		(*-----------------------Weiterschaltbedingungen----------------------------*)
		IF zyl_bawe_vorschub.st_ctrl.out.b_ausgefahren AND gb_ba_auto_kontroller THEN
			zyl_bawe_vorschub.st_ctrl.in.b_ausfahren := FALSE;
			IF i16_akt_einfaedeln < i16_vorgabe_einfaedeln THEN
				fb_state_entry.i16_next_step := 640;
			ELSE
				fb_state_entry.i16_next_step := 690; (*mit Wartezeit alt auf 700*)
			END_IF
		END_IF

(*=======================================================*)
	640:	(* Halter links ausfahren *)
		IF fb_state_entry.E THEN
			zyl_bawe_halter_li.st_ctrl.in.b_ausfahren := TRUE;
		END_IF

		(*-----------------------Weiterschaltbedingungen----------------------------*)
		IF zyl_bawe_halter_li.st_ctrl.out.b_ausgefahren AND gb_ba_auto_kontroller THEN
			zyl_bawe_halter_li.st_ctrl.in.b_ausfahren := FALSE;
			fb_state_entry.i16_next_step := 650;
		END_IF

(*=======================================================*)
	650:	(* Fänger links einfahren *)
		IF fb_state_entry.E THEN
			zyl_bawe_faenger_li.st_ctrl.in.b_einfahren := TRUE;
		END_IF

		(*-----------------------Weiterschaltbedingungen----------------------------*)
		IF zyl_bawe_faenger_li.st_ctrl.out.b_eingefahren AND gb_ba_auto_kontroller THEN
			zyl_bawe_faenger_li.st_ctrl.in.b_einfahren := FALSE;
			fb_state_entry.i16_next_step := 660;
		END_IF

(*=======================================================*)
	660:	(* Vorschub einfahren *)
		IF fb_state_entry.E THEN
			zyl_bawe_vorschub.st_ctrl.in.b_einfahren := TRUE;
		END_IF

		(*-----------------------Weiterschaltbedingungen----------------------------*)
		IF zyl_bawe_vorschub.st_ctrl.out.b_eingefahren AND gb_ba_auto_kontroller THEN
			zyl_bawe_vorschub.st_ctrl.in.b_einfahren := FALSE;
			fb_state_entry.i16_next_step := 670;
		END_IF

(*=======================================================*)
	670:	(* Fänger links ausfahren *)
		IF fb_state_entry.E THEN
			zyl_bawe_faenger_li.st_ctrl.in.b_ausfahren := TRUE;
		END_IF

		(*-----------------------Weiterschaltbedingungen----------------------------*)
		IF zyl_bawe_faenger_li.st_ctrl.out.b_ausgefahren AND gb_ba_auto_kontroller THEN
			zyl_bawe_faenger_li.st_ctrl.in.b_ausfahren := FALSE;
			fb_state_entry.i16_next_step := 680;
		END_IF

(*=======================================================*)
	680:	(* Halter links einfahren *)
		IF fb_state_entry.E THEN
			zyl_bawe_halter_li.st_ctrl.in.b_einfahren := TRUE;
		END_IF

		(*-----------------------Weiterschaltbedingungen----------------------------*)
		IF zyl_bawe_halter_li.st_ctrl.out.b_eingefahren AND gb_ba_auto_kontroller THEN
			zyl_bawe_halter_li.st_ctrl.in.b_einfahren := FALSE;
			fb_state_entry.i16_next_step := 630;
		END_IF
(*=======================================================*)
	690:	(* Wartezeit damit der Fänger vom WZ trifft*)
		IF	 fb_state_entry.E THEN
			fb_ton_wz.IN:=FALSE;
		END_IF
		fb_ton_wz(IN:=TRUE,PT:=t#1000ms);
		(*-----------------------Weiterschaltbedingungen----------------------------*)
		IF 	fb_ton_wz.Q THEN
			fb_ton_wz.IN:=FALSE;
			fb_state_entry.i16_next_step := 700;
		END_IF

(*=======================================================*)
	700:	(* Nocken für Zylinder am Bandeinzug einschalten und somit Bandfänger ausfahren bzw. Bremse an Servobandeinzug wieder fest machen. *)
		CASE gst_datensatz.st_wkz.i16_typ_bandeinzug OF

			BANDWECHSLER_V2:

				IF fb_state_entry.E THEN
					(* Bandwechsler V2 ohne Sensoren und anderen Zylindern *)
					gst_datensatz.st_wkz.nockenschaltwerk_bestueckachse.arr_nocken[NO_BW_BANDFAENGER_BAWEV2_EINFAHREN].b_camvalid := TRUE;
					gst_datensatz.st_wkz.nockenschaltwerk_bestueckachse.arr_nocken[NO_BW_BANDFAENGER_BAWEV2_AUSFAHREN].b_camvalid := TRUE;
					gst_datensatz.st_wkz.nockenschaltwerk_bestueckachse.arr_nocken[NO_BW_BANDKLEMMEN_BAWEV2_EINFAHREN].b_camvalid := TRUE;
					gst_datensatz.st_wkz.nockenschaltwerk_bestueckachse.arr_nocken[NO_BW_BANDKLEMMEN_BAWEV2_AUSFAHREN].b_camvalid := TRUE;

					gst_datensatz.st_wkz.nockenschaltwerk_bestueckachse.arr_nocken[NO_PNEUMATIKBANDEINZUG_GLS].b_camvalid := TRUE;

					zyl_bandfaenger.fb.b_no_gesteuert_im_norm_betrieb := FALSE;
					zyl_bandklemmen.fb.b_no_gesteuert_im_norm_betrieb := FALSE;
					fb_ton_wz.PT := t#500ms;
					fb_ton_wz.IN := TRUE;
				END_IF
		
				(*-----------------------Weiterschaltbedingungen----------------------------*)
				IF fb_ton_wz.Q THEN
					fb_ton_wz.IN := FALSE;
					fb_state_entry.i16_next_step := 710;
				END_IF

			SERVO:
				IF fb_state_entry.E THEN
					axis_bandeinzug_achse.st_ctrl.in.b_bremse_auf := TRUE;	(* Bremse auf zum Position übernehmen *)
				END_IF

				(*-----------------------Weiterschaltbedingungen----------------------------*)
				IF axis_bandeinzug_achse.st_ctrl.out.b_bremse_geoeffnet THEN
					axis_bandeinzug_achse.st_ctrl.in.b_bremse_auf := FALSE;
					fb_state_entry.i16_next_step := 710;
				END_IF
		END_CASE;

(*=======================================================*)
	710:	(* Fänger links einfahren *)
		IF fb_state_entry.E THEN
			zyl_bawe_faenger_li.st_ctrl.in.b_einfahren := TRUE;
		END_IF

		(*-----------------------Weiterschaltbedingungen----------------------------*)
		IF zyl_bawe_faenger_li.st_ctrl.out.b_eingefahren
		AND gb_ba_auto_kontroller THEN
			zyl_bawe_faenger_li.st_ctrl.in.b_einfahren := FALSE;
			(* Bandwechsel ist fertig *)
			st_ctrl_out.b_fertig := TRUE;
			fb_state_entry.i16_next_step := BEREIT;
		END_IF

(*=======================================================*)
	FEHLER:
		IF fb_state_entry.E THEN
			st_ctrl_out.b_fehler := TRUE;
			fb_ton_quitt.IN := FALSE;
			zyl_bawe_vorschub.st_ctrl.in.b_quittieren := FALSE;
			zyl_bawe_querschub.st_ctrl.in.b_quittieren := FALSE;
			zyl_bawe_faenger_li.st_ctrl.in.b_quittieren := FALSE;
			zyl_bawe_faenger_re.st_ctrl.in.b_quittieren := FALSE;
			zyl_bawe_halter_li.st_ctrl.in.b_quittieren := FALSE;
			zyl_bawe_halter_re.st_ctrl.in.b_quittieren := FALSE;
			zyl_haspel_verschieben.st_ctrl.in.b_quittieren := FALSE;
			zyl_bandeinzuege_verschieben.st_ctrl.in.b_quittieren := FALSE;
		END_IF

		(*-----------------------Weiterschaltbedingungen----------------------------*)
		IF st_ctrl_in.b_quitt AND NOT fb_state_entry.E THEN
			st_ctrl_out.b_fehler := TRUE;
			zyl_bawe_vorschub.st_ctrl.in.b_quittieren := TRUE;
			zyl_bawe_querschub.st_ctrl.in.b_quittieren := TRUE;
			zyl_bawe_faenger_li.st_ctrl.in.b_quittieren := TRUE;
			zyl_bawe_faenger_re.st_ctrl.in.b_quittieren := TRUE;
			zyl_bawe_halter_li.st_ctrl.in.b_quittieren := TRUE;
			zyl_bawe_halter_re.st_ctrl.in.b_quittieren := TRUE;
			zyl_haspel_verschieben.st_ctrl.in.b_quittieren := TRUE;
			zyl_bandeinzuege_verschieben.st_ctrl.in.b_quittieren := TRUE;
			fb_ton_quitt.IN := TRUE;
		END_IF

		IF fb_ton_quitt.Q THEN
			fb_ton_quitt.IN := FALSE;
			fb_state_entry.i16_next_step := INIT;
		END_IF

(*=======================================================*)
	STOP:
		IF fb_state_entry.E THEN
			fb_ton_quitt.IN := FALSE;
			zyl_bawe_vorschub.st_ctrl.in.b_quittieren := FALSE;
			zyl_bawe_querschub.st_ctrl.in.b_quittieren := FALSE;
			zyl_bawe_faenger_li.st_ctrl.in.b_quittieren := FALSE;
			zyl_bawe_faenger_re.st_ctrl.in.b_quittieren := FALSE;
			zyl_bawe_halter_li.st_ctrl.in.b_quittieren := FALSE;
			zyl_bawe_halter_re.st_ctrl.in.b_quittieren := FALSE;
			zyl_haspel_verschieben.st_ctrl.in.b_quittieren := FALSE;
			zyl_bandeinzuege_verschieben.st_ctrl.in.b_quittieren := FALSE;
		END_IF

		(*-----------------------Weiterschaltbedingungen----------------------------*)
		IF st_ctrl_in.b_quitt AND NOT fb_state_entry.E THEN
			fb_ton_quitt.IN := TRUE;
			zyl_bawe_vorschub.st_ctrl.in.b_quittieren := TRUE;
			zyl_bawe_querschub.st_ctrl.in.b_quittieren := TRUE;
			zyl_bawe_faenger_li.st_ctrl.in.b_quittieren := TRUE;
			zyl_bawe_faenger_re.st_ctrl.in.b_quittieren := TRUE;
			zyl_bawe_halter_li.st_ctrl.in.b_quittieren := TRUE;
			zyl_bawe_halter_re.st_ctrl.in.b_quittieren := TRUE;
			zyl_haspel_verschieben.st_ctrl.in.b_quittieren := TRUE;
			zyl_bandeinzuege_verschieben.st_ctrl.in.b_quittieren := TRUE;
		END_IF

		IF fb_ton_quitt.Q THEN
			fb_ton_quitt.IN := FALSE;
			fb_state_entry.i16_next_step := INIT;
		END_IF
END_CASE

fb_state_entry(
	i16_next_step:= , 
	i16_pos:= 2,
	s_debugtext:= ,
	E=> ,
	X=> , 
	i16_step=> ,
	i16_last_step=> );

IF st_config.b_config_fertig THEN
	(* Fehlermeldungen und Betriebsmeldungen ab dem Startindex in die globalen Meldungsarrays schreiben *)
	garr_stoermeldungen[st_config.i16_meld_startindex + 0] := sm_halter_nicht_oben;
	garr_stoermeldungen[st_config.i16_meld_startindex + 1] := sm_bandwechsel_ohne_ende;
	garr_stoermeldungen[st_config.i16_meld_startindex + 2] := sm_kein_band_anderer_einzug;
	garr_stoermeldungen[st_config.i16_meld_startindex + 3] := sm_kein_band_in_akt_einzug;
	garr_stoermeldungen[st_config.i16_meld_startindex + 4] := FALSE;
	garr_stoermeldungen[st_config.i16_meld_startindex + 5] := FALSE;
	garr_stoermeldungen[st_config.i16_meld_startindex + 6] := FALSE;
	garr_stoermeldungen[st_config.i16_meld_startindex + 7] := FALSE;
	garr_stoermeldungen[st_config.i16_meld_startindex + 8] := FALSE;
	garr_stoermeldungen[st_config.i16_meld_startindex + 9] := FALSE;
	garr_stoermeldungen[st_config.i16_meld_startindex + 10] := FALSE;
	garr_stoermeldungen[st_config.i16_meld_startindex + 11] := FALSE;
	garr_stoermeldungen[st_config.i16_meld_startindex + 12] := FALSE;
	garr_stoermeldungen[st_config.i16_meld_startindex + 13] := FALSE;
	garr_stoermeldungen[st_config.i16_meld_startindex + 14] := FALSE;
	garr_stoermeldungen[st_config.i16_meld_startindex + 15] := FALSE;
	garr_stoermeldungen[st_config.i16_meld_startindex + 16] := FALSE;
	garr_stoermeldungen[st_config.i16_meld_startindex + 17] := FALSE;
	garr_stoermeldungen[st_config.i16_meld_startindex + 18] := FALSE;
	garr_stoermeldungen[st_config.i16_meld_startindex + 19] := FALSE;
	
	garr_betriebsmeldungen[st_config.i16_meld_startindex + 0] := bm_bandwechselvorgang;
	garr_betriebsmeldungen[st_config.i16_meld_startindex + 1] := bm_bandwechsel_manuell;
	garr_betriebsmeldungen[st_config.i16_meld_startindex + 2] := FALSE;
	garr_betriebsmeldungen[st_config.i16_meld_startindex + 3] := FALSE;
	garr_betriebsmeldungen[st_config.i16_meld_startindex + 4] := FALSE;
	garr_betriebsmeldungen[st_config.i16_meld_startindex + 5] := FALSE;
	garr_betriebsmeldungen[st_config.i16_meld_startindex + 6] := FALSE;
	garr_betriebsmeldungen[st_config.i16_meld_startindex + 7] := FALSE;
	garr_betriebsmeldungen[st_config.i16_meld_startindex + 8] := FALSE;
	garr_betriebsmeldungen[st_config.i16_meld_startindex + 9] := FALSE;
	garr_betriebsmeldungen[st_config.i16_meld_startindex + 10] := FALSE;
	garr_betriebsmeldungen[st_config.i16_meld_startindex + 11] := FALSE;
	garr_betriebsmeldungen[st_config.i16_meld_startindex + 12] := FALSE;
	garr_betriebsmeldungen[st_config.i16_meld_startindex + 13] := FALSE;
	garr_betriebsmeldungen[st_config.i16_meld_startindex + 14] := FALSE;
	garr_betriebsmeldungen[st_config.i16_meld_startindex + 15] := FALSE;
	garr_betriebsmeldungen[st_config.i16_meld_startindex + 16] := FALSE;
	garr_betriebsmeldungen[st_config.i16_meld_startindex + 17] := FALSE;
	garr_betriebsmeldungen[st_config.i16_meld_startindex + 18] := FALSE;
	garr_betriebsmeldungen[st_config.i16_meld_startindex + 19] := FALSE;
END_IF
END_PROGRAM

(* POU Maschine1700/Einpresskraftueberwachung/ST_Einpress_Kontroller, ST *)
PROGRAM ST_Einpress_Kontroller
VAR_INPUT
	st_config									: struct_config;
	st_ctrl_in									: struct_ctrl_in;
	lr_achsposition							: LREAL;
END_VAR
VAR_IN_OUT
	st_visu									: struct_visu;
	st_einpressen							: struct_einpresskraftueberwachung;
END_VAR
VAR_OUTPUT
	st_ctrl_out								: struct_ctrl_out;
END_VAR
VAR
	fb_ton_wz								: TON;
	fb_ton_uez								: TON;
	fb_ton_quitt								: TON;
	fb_r_trig_start								: R_TRIG;
	fb_f_trig_bestueckposzaehler				: F_TRIG;
	fb_state_entry								: ST_StateEntry;
	lr_kraft_n									: LREAL := 0.0;
	i16_pin_nr								: INT := 0;
	i16_pin_nr_alt								: INT := 0;
	i16_kraftfaktor								: INT := 0;
	sm_fehler_einpressmodus					: BOOL := FALSE;
	sm_aktkraft_groesser_maxkraft_einpressen	: BOOL := FALSE;
	sm_aktkraft_groesserr_mittelkraft_einpressen	: BOOL := FALSE;
	sm_fehler_analogwert_kraftmessdose		: BOOL := FALSE;
	sm_max_mb_ueberschritten					: BOOL := FALSE;
	sm_max_einstell_mb_ueberschritten			: BOOL := FALSE;

	a_start_messung							AT %Q* : BOOL := FALSE;
	a_messbereich_1_oder_2					AT %Q* : BOOL := FALSE;	(* MB1 = low, MB2 = high *)

	st_ausgabe								: struct_einpressausgabe;
	lr_vergleich_kraft_einpressen				: LREAL;
	lr_arr_aktuelle_kraft						: ARRAY[0..9] OF LREAL;
	lr_max_kraft_im_arr						: LREAL;
	lr_mittel_kraft_im_arr						: LREAL;
	lr_aktuelle_kraft_pin						: LREAL;
	lr_akutelle_kraft_messbereich			: LREAL;
	i										: INT;
	b_ueberwachung_gueltig					: BOOL;
END_VAR
VAR CONSTANT
	i_KRAFTFAKTOR_MB1		: INT := 200;	(* Der Kraftfaktor richtet sich nach der Messbereichskalibrierung in der Zusatzsoftware (ICAM) für den Ladungsverstärker *)
	i_KRAFTFAKTOR_MB2		: INT := 2000;
END_VAR
(* Zeiten *)
fb_ton_wz(IN:= , PT:= , Q=>  , ET=> );
fb_ton_uez(IN:= , PT:= , Q=>  , ET=> );

fb_ton_quitt(IN:= , PT:= t#100ms, Q=> , ET=> );

(* Flanken *)
fb_r_trig_start(CLK:= st_ctrl_in.b_start, Q=> );
fb_f_trig_bestueckposzaehler(CLK:= nockenschaltwerk_bestueckachse.fb.arr_spur[SP_BESTUECKSCHIEBERHUB ], Q=> );

(* Analogwert Kraftmessdose *)
kraftmessdose.fb(
	t_verzoegerung:= t#500ms,
	st_config:= kraftmessdose.fb.st_config);

(* Berechnung der aktuellen Kraft in Newton aus dem Analogwert in  Volt. *)
(* Die Normierung der Analogspannung als Kraft erfolgt mit dem Kalibrierschein der Kraftmessdose und der Software "ICAM5073" *)
(* Eingestellter Messbereich1: 0 - 200N, Messbereich2: 0 - 2000N *)
IF a_messbereich_1_oder_2 THEN
	i16_kraftfaktor := i_KRAFTFAKTOR_MB2;
ELSE
	i16_kraftfaktor := i_KRAFTFAKTOR_MB1;
END_IF

(* Behandlung Ausnahmefall Division durch 0  *)
IF kraftmessdose.fb.i16_anzeigewert_max <> 0 THEN
	lr_kraft_n := i16_kraftfaktor * kraftmessdose.fb.st_sensor.e_i16_value / kraftmessdose.fb.i16_anzeigewert_max;
END_IF

(* ===============Toplevel================ *)
IF fb_state_entry.i16_next_step > INIT AND fb_state_entry.i16_next_step < FEHLER THEN
	IF fb_state_entry.i16_next_step < STOP THEN
		IF st_ctrl_in.b_stop THEN
			fb_state_entry.i16_next_step := STOP;
		END_IF
	END_IF

	(* Fehlersignal der Kraftmessdose *)
	IF st_config.b_station_aktiv THEN
		IF kraftmessdose.fb.b_error THEN
			sm_fehler_analogwert_kraftmessdose := TRUE;
			fb_state_entry.i16_next_step := FEHLER;
		END_IF
		IF 	(NOT a_messbereich_1_oder_2 AND lr_kraft_n > i_KRAFTFAKTOR_MB1) OR
			(a_messbereich_1_oder_2 AND lr_kraft_n > i_KRAFTFAKTOR_MB2) OR
			(gst_datensatz.st_band.st_einpressen.st_einstellungen.lr_maxkraft_einpressen > i_KRAFTFAKTOR_MB2)
			THEN
				sm_max_mb_ueberschritten := TRUE;
				fb_state_entry.i16_next_step := FEHLER;
		END_IF
		IF gst_datensatz.st_band.st_einpressen.st_einstellungen.lr_maxkraft_einpressen > i_KRAFTFAKTOR_MB2 THEN
			sm_max_einstell_mb_ueberschritten := TRUE;
			fb_state_entry.i16_next_step := FEHLER;
		END_IF
	END_IF
END_IF

(* ======================================Schrittkette======================================== *)
fb_state_entry(
	i16_next_step:= ,
	i16_pos:= 1,
	s_debugtext:= ,
	E=> ,
	X=> ,
	i16_step=> ,
	i16_last_step=> );

CASE fb_state_entry.i16_step OF
(*=======================================================*)
	INIT_OBJ:
		IF st_config.b_config_fertig THEN
			a_messbereich_1_oder_2 := FALSE;
			fb_state_entry.i16_next_step := INIT;
		END_IF

(*=======================================================*)
	INIT:
		IF fb_state_entry.E THEN
			fb_ton_wz.IN := FALSE;
			fb_ton_uez.IN := FALSE;
			fb_ton_quitt.IN := FALSE;
			st_ctrl_out.b_fehler := FALSE;
			st_ctrl_out.b_bereit := FALSE;
			st_ctrl_out.b_fertig := FALSE;
			a_start_messung := FALSE;
			b_ueberwachung_gueltig := FALSE;
			i16_pin_nr := 0;
			sm_fehler_einpressmodus := FALSE;
			sm_aktkraft_groesser_maxkraft_einpressen := FALSE;
			sm_aktkraft_groesserr_mittelkraft_einpressen := FALSE;
			sm_fehler_analogwert_kraftmessdose := FALSE;
			sm_max_mb_ueberschritten := FALSE;
			sm_max_einstell_mb_ueberschritten := FALSE;
			(*Löschen der gesammelten Kräfte der letzten zehn Hübe*)
			FOR i := 0 TO 9 DO
				lr_arr_aktuelle_kraft[i] := 0;
			END_FOR

		END_IF

		(*-----------------------Weiterschaltbedingungen----------------------------*)
		IF st_ctrl_in.b_init THEN
			fb_state_entry.i16_next_step := BEREIT;
		END_IF

(*=======================================================*)
	BEREIT:
		IF fb_state_entry.E THEN
			st_ctrl_out.b_bereit := TRUE;
			st_ctrl_out.b_fertig := TRUE;
			i16_pin_nr := 0;
			i16_pin_nr_alt := 0;
		END_IF

		(*-----------------------Weiterschaltbedingungen----------------------------*)
		IF st_ctrl_in.b_start THEN
			fb_state_entry.i16_next_step := 110;
		END_IF

(*=======================================================*)
	110:	(* Kraftmessung starten *)
		IF fb_state_entry.E THEN
			st_ctrl_out.b_fertig := FALSE;
			a_start_messung := TRUE;
			st_ausgabe.st_ergebnisse.lr_maxkraft_einpressen := 0;
			st_ausgabe.st_ergebnisse.lr_maxkraft_einpres_proHub:=0;
			st_ausgabe.st_ergebnisse.lr_ueberlaufkraft := 0;
			lr_aktuelle_kraft_pin := 0;
			lr_akutelle_kraft_messbereich := 0;
		END_IF

		(* Hochzählen mit der Anzahl der bestückten Pins *)
		IF fb_f_trig_bestueckposzaehler.Q THEN
			i16_pin_nr := i16_pin_nr +1;
		END_IF

		(*aktuell höchste Kraft wird sich gemerkt*)
		IF  lr_kraft_n > lr_aktuelle_kraft_pin THEN
			lr_aktuelle_kraft_pin := lr_kraft_n;
			lr_akutelle_kraft_messbereich := lr_kraft_n;
		END_IF

		(*Bei jedem neuen Pin wird die höchste gemessene Kraft in ein Array geschrieben und die älteste von den letzten 10
		wird gelöscht*)
		IF i16_pin_nr_alt <> i16_pin_nr AND ST_Virtuelle_Masterachse.i16_bestueckachse_cam_table_id = 5 THEN
			FOR i:=9 TO 1 BY -1 DO
				lr_arr_aktuelle_kraft[i]:=lr_arr_aktuelle_kraft[i-1];
			END_FOR
			lr_arr_aktuelle_kraft[0] := lr_aktuelle_kraft_pin;
			lr_aktuelle_kraft_pin := 0;
			i16_pin_nr_alt := i16_pin_nr;
		END_IF

		(*Überprüfung, ob das Array komplett mit Werten befüllt ist*)
		FOR i := 0 TO 9 DO
			IF lr_arr_aktuelle_kraft[i] = 0 THEN
				b_ueberwachung_gueltig := FALSE;
				EXIT;
			ELSE
				b_ueberwachung_gueltig := TRUE;
			END_IF
		END_FOR

		(*Auswahl Auswertemodus*)
		CASE st_einpressen.st_einstellungen.enu_modus OF

			KEIN_MODUS:	(* Kraftübwerachung ausgeschalten *)
					;
			F_MAXWERT:	(* Einpressen mit Überwachung auf den Maximalwert *)

				IF b_ueberwachung_gueltig THEN
					lr_max_kraft_im_arr := 0;
					(*Maximalkraft im Array wird gesucht*)
					FOR i := 0 TO 9 DO
						IF  lr_arr_aktuelle_kraft[i] > lr_max_kraft_im_arr THEN
							lr_max_kraft_im_arr := lr_arr_aktuelle_kraft[i];
						END_IF
					END_FOR

					(* nur bei voller Drehzahl und normalen Bestückbild mit ermittelter Kraft prüfen*)
					IF ST_TippTasten.i16_akt_stufe = 9 AND (FIND(gst_datensatz.st_md.s_aktuelle_artikelnummer,'ruef') = 0		(*es wird nur auf ruef abgefragt, weil das P groß oder klein sein kann*)
						 AND FIND(gst_datensatz.st_md.s_aktuelle_artikelnummer,'erth') = 0) THEN
						lr_vergleich_kraft_einpressen:=lr_max_kraft_im_arr;
					ELSE
						lr_vergleich_kraft_einpressen:=800;
					END_IF

					(* Fehlerfall: Ermittelte Maximalkraft überschritten nur im Automatik Betrieb *)
					IF  gi16_betriebsart = AUTO AND lr_kraft_n > lr_vergleich_kraft_einpressen + st_einpressen.st_einstellungen.lr_delta_kraft THEN
						st_einpressen.st_einstellungen.lr_maxkraft_einpressen := lr_kraft_n;
						st_ausgabe.st_ergebnisse.lr_maxkraft_einpressen:=lr_kraft_n;
						sm_aktkraft_groesser_maxkraft_einpressen := TRUE;
						fb_state_entry.i16_next_step := FEHLER;
					END_IF
				END_IF


			F_MITTELWERT:	(* Einpressen mit Überwachung auf den Mittelwert *)

				IF b_ueberwachung_gueltig THEN
					(*Kraft im Array wird aufaddiert*)
					FOR i := 0 TO 9 DO
						lr_mittel_kraft_im_arr := lr_mittel_kraft_im_arr + lr_arr_aktuelle_kraft[i];
					END_FOR
					(*Mittelwert der Kräfte im Array wird gebildet*)
					lr_mittel_kraft_im_arr := lr_mittel_kraft_im_arr / 10;

					(* nur bei voller Drehzahl und normalen Bestückbild mit ermittelter Kraft prüfen*)
					IF ST_TippTasten.i16_akt_stufe = 9 AND (FIND(gst_datensatz.st_md.s_aktuelle_artikelnummer,'ruef') = 0			(*es wird nur auf ruef abgefragt, weil das P groß oder klein sein kann*)
						AND FIND(gst_datensatz.st_md.s_aktuelle_artikelnummer,'erth') = 0) THEN
						lr_vergleich_kraft_einpressen:=lr_mittel_kraft_im_arr;
					ELSE
						lr_vergleich_kraft_einpressen:=800;
					END_IF

					(* Fehlerfall: Ermittelte Maximalkraft überschritten nur im Automatik Betrieb *)
					IF  gi16_betriebsart = AUTO AND lr_kraft_n > lr_vergleich_kraft_einpressen + st_einpressen.st_einstellungen.lr_delta_kraft THEN
						sm_aktkraft_groesserr_mittelkraft_einpressen := TRUE;
						st_einpressen.st_einstellungen.lr_maxkraft_einpressen := lr_kraft_n;
						st_ausgabe.st_ergebnisse.lr_maxkraft_einpressen:=lr_kraft_n;
						fb_state_entry.i16_next_step := FEHLER;
					END_IF
				END_IF
		END_CASE

		(* Manuelle Messbereichsumschaltung anhand des Einstellwertes für Maximalkraft beim Einpressen. *)
		IF gst_datensatz.st_band.st_einpressen.st_einstellungen.lr_maxkraft_einpressen > (i_KRAFTFAKTOR_MB1 * 0.75) THEN
			a_messbereich_1_oder_2 := TRUE;
		ELSE
			(* Automatische Messbereichsumschaltung, wenn die maximale Einpresskraft 75% des Messbereichsendwertes überschreitet. *)
			IF lr_akutelle_kraft_messbereich > (i_KRAFTFAKTOR_MB1 * 0.75) THEN
				a_messbereich_1_oder_2 := TRUE;
			END_IF
		END_IF

		(*-----------------------Weiterschaltbedingungen----------------------------*)
		IF NOT st_ctrl_in.b_start THEN
			(* Messbereichsanpassung nur, wenn die Krafteinstellung für maximale Einpresskraft es erlaubt. *)
			IF gst_datensatz.st_band.st_einpressen.st_einstellungen.lr_maxkraft_einpressen < (i_KRAFTFAKTOR_MB1 * 0.75) THEN
				(* Automatische Messbereichsumschaltung, wenn die maximale Einpresskraft 50% des Messbereichsendwertes unterschreitet. *)
				IF lr_akutelle_kraft_messbereich < (i_KRAFTFAKTOR_MB1 * 0.5) THEN
					a_messbereich_1_oder_2 := FALSE;
				END_IF
			END_IF
			a_start_messung := FALSE;
			fb_state_entry.i16_next_step := BEREIT;
		END_IF

(*=======================================================*)
	FEHLER:
		IF fb_state_entry.E THEN
			st_ctrl_out.b_fehler := TRUE;
			fb_ton_quitt.IN := FALSE;
		END_IF

		(* Aufzeichnen der Überlaufkraft nach einem Einpressfehler *)
		IF  lr_kraft_n > st_ausgabe.st_ergebnisse.lr_ueberlaufkraft THEN
			st_ausgabe.st_ergebnisse.lr_ueberlaufkraft := lr_kraft_n;
		END_IF

		(*-----------------------Weiterschaltbedingungen----------------------------*)
		IF st_ctrl_in.b_quitt AND NOT fb_state_entry.E THEN
			st_ctrl_out.b_fehler := FALSE;
			fb_ton_quitt.IN := TRUE;
		END_IF

		IF fb_ton_quitt.Q THEN
			fb_ton_quitt.IN := FALSE;
			fb_state_entry.i16_next_step := INIT;
		END_IF

(*=======================================================*)
	STOP:
		IF fb_state_entry.E THEN
			fb_ton_quitt.IN := FALSE;
		END_IF

		(*-----------------------Weiterschaltbedingungen----------------------------*)
		IF st_ctrl_in.b_quitt AND NOT fb_state_entry.E THEN
			fb_ton_quitt.IN := TRUE;
		END_IF

		IF fb_ton_quitt.Q THEN
			fb_ton_quitt.IN := FALSE;
			fb_state_entry.i16_next_step := INIT;
		END_IF
END_CASE

fb_state_entry(
	i16_next_step:= ,
	i16_pos:= 2,
	s_debugtext:= ,
	E=> ,
	X=> ,
	i16_step=> ,
	i16_last_step=> );

(* Fehlermeldungen und Betriebsmeldungen ab dem Startindex in die globalen Meldungsarrays schreiben *)
garr_stoermeldungen[st_config.i16_meld_startindex + 0] := sm_fehler_einpressmodus;
garr_stoermeldungen[st_config.i16_meld_startindex + 1] := sm_aktkraft_groesser_maxkraft_einpressen;
garr_stoermeldungen[st_config.i16_meld_startindex + 2] := sm_aktkraft_groesserr_mittelkraft_einpressen;
garr_stoermeldungen[st_config.i16_meld_startindex + 3] := sm_fehler_analogwert_kraftmessdose;
garr_stoermeldungen[st_config.i16_meld_startindex + 4] := sm_max_mb_ueberschritten;
garr_stoermeldungen[st_config.i16_meld_startindex + 5] := sm_max_einstell_mb_ueberschritten;
garr_stoermeldungen[st_config.i16_meld_startindex + 6] := FALSE;
garr_stoermeldungen[st_config.i16_meld_startindex + 7] := FALSE;
garr_stoermeldungen[st_config.i16_meld_startindex + 8] := FALSE;
garr_stoermeldungen[st_config.i16_meld_startindex + 9] := FALSE;
garr_stoermeldungen[st_config.i16_meld_startindex + 10] := FALSE;
garr_stoermeldungen[st_config.i16_meld_startindex + 11] := FALSE;
garr_stoermeldungen[st_config.i16_meld_startindex + 12] := FALSE;
garr_stoermeldungen[st_config.i16_meld_startindex + 13] := FALSE;
garr_stoermeldungen[st_config.i16_meld_startindex + 14] := FALSE;
garr_stoermeldungen[st_config.i16_meld_startindex + 15] := FALSE;
garr_stoermeldungen[st_config.i16_meld_startindex + 16] := FALSE;
garr_stoermeldungen[st_config.i16_meld_startindex + 17] := FALSE;
garr_stoermeldungen[st_config.i16_meld_startindex + 18] := FALSE;
garr_stoermeldungen[st_config.i16_meld_startindex + 19] := FALSE;

garr_betriebsmeldungen[st_config.i16_meld_startindex + 0] := FALSE;
garr_betriebsmeldungen[st_config.i16_meld_startindex + 1] := FALSE;
garr_betriebsmeldungen[st_config.i16_meld_startindex + 2] := FALSE;
garr_betriebsmeldungen[st_config.i16_meld_startindex + 3] := FALSE;
garr_betriebsmeldungen[st_config.i16_meld_startindex + 4] := FALSE;
garr_betriebsmeldungen[st_config.i16_meld_startindex + 5] := FALSE;
garr_betriebsmeldungen[st_config.i16_meld_startindex + 6] := FALSE;
garr_betriebsmeldungen[st_config.i16_meld_startindex + 7] := FALSE;
garr_betriebsmeldungen[st_config.i16_meld_startindex + 8] := FALSE;
garr_betriebsmeldungen[st_config.i16_meld_startindex + 9] := FALSE;
garr_betriebsmeldungen[st_config.i16_meld_startindex + 10] := FALSE;
garr_betriebsmeldungen[st_config.i16_meld_startindex + 11] := FALSE;
garr_betriebsmeldungen[st_config.i16_meld_startindex + 12] := FALSE;
garr_betriebsmeldungen[st_config.i16_meld_startindex + 13] := FALSE;
garr_betriebsmeldungen[st_config.i16_meld_startindex + 14] := FALSE;
garr_betriebsmeldungen[st_config.i16_meld_startindex + 15] := FALSE;
garr_betriebsmeldungen[st_config.i16_meld_startindex + 16] := FALSE;
garr_betriebsmeldungen[st_config.i16_meld_startindex + 17] := FALSE;
garr_betriebsmeldungen[st_config.i16_meld_startindex + 18] := FALSE;
garr_betriebsmeldungen[st_config.i16_meld_startindex + 19] := FALSE;
END_PROGRAM

(* POU Maschine1700/Band/ST_Bandeinzug_Kontroller_1700, ST *)
PROGRAM ST_Bandeinzug_Kontroller_1700
VAR_INPUT
	st_config						: struct_config;
	st_ctrl_in						: struct_ctrl_in;
END_VAR
VAR_IN_OUT
	st_visu						: struct_visu;
END_VAR
VAR_OUTPUT
	st_ctrl_out					: struct_ctrl_out;
END_VAR
VAR
	fb_ton_wz					: TON;
	fb_ton_uez					: TON;
	fb_ton_quitt					: TON;
	fb_state_entry					: ST_StateEntry;
	b_einzug_stop				: BOOL := FALSE;

	fb_r_trig_vorschubkontrolle		: R_TRIG;
	fb_f_trig_vorschubkontrolle		: F_TRIG;
	fb_r_trig_nocke_einzug			: R_TRIG;
	fb_f_trig_nocke_einzug			: F_TRIG;
	b_hm_pos_flanke_vorschub	: BOOL := FALSE;
	b_hm_neg_flanke_vorschub	: BOOL := FALSE;
	sm_fehler_bandvorschub		: BOOL := FALSE;
	sm_keine_busverbindung	: BOOL := FALSE;

	e_wc_state					AT %I* : BOOL;	(* 0=Data valid, 1=Data invalid *)
	e_gls_bandvorschubkontrolle	AT %I* : BOOL;
END_VAR
(* Zeiten *)
fb_ton_wz(IN:= , PT:= , Q=>  , ET=> );
fb_ton_uez(IN:= , PT:= , Q=>  , ET=> );
fb_ton_quitt(IN:= , PT:= t#100ms, Q=> , ET=> );

(* Flanken *)
fb_f_trig_vorschubkontrolle(CLK:= e_gls_bandvorschubkontrolle, Q=> );
fb_r_trig_vorschubkontrolle(CLK:= e_gls_bandvorschubkontrolle, Q=> );
fb_f_trig_nocke_einzug(CLK:= nockenschaltwerk_bestueckachse.fb.arr_spur[SP_PNEUMATIKBANDEINZUG_GLS], Q=> );
fb_r_trig_nocke_einzug(CLK:= nockenschaltwerk_bestueckachse.fb.arr_spur[SP_PNEUMATIKBANDEINZUG_GLS], Q=> );

(* Toplevel *)
IF fb_state_entry.i16_next_step > INIT AND fb_state_entry.i16_next_step < FEHLER THEN
	IF fb_state_entry.i16_next_step < STOP THEN
		IF st_ctrl_in.b_stop THEN
			fb_state_entry.i16_next_step := STOP;
		END_IF
	END_IF
	(* Allgemeine Fehler *)
	IF	NOT gst_datensatz.st_md.b_wt_transport_simulation AND
		(zyl_bandfaenger.st_ctrl.out.b_fehler OR
		zyl_bandklemmen.st_ctrl.out.b_fehler)
		 THEN
			fb_state_entry.i16_next_step := FEHLER;

	(* Zylinder im Handbetrieb *)
	ELSIF	 gi16_betriebsart = HAND AND (
			(st_visu.st_zyl.i16_nr_zyl_im_handbetrieb = zyl_bandfaenger.fb.st_config.i16_identnummer) OR
			(st_visu.st_zyl.i16_nr_zyl_im_handbetrieb = zyl_bandklemmen.fb.st_config.i16_identnummer) )
			THEN
			fb_state_entry.i16_next_step := FEHLER;
	END_IF
END_IF

(* ======================================Schrittkette======================================== *)
fb_state_entry(
	i16_next_step:= , 
	i16_pos:= 1,
	s_debugtext:= ,
	E=> ,
	X=> , 
	i16_step=> ,
	i16_last_step=> );

CASE fb_state_entry.i16_step OF
(*=======================================================*)
	INIT_OBJ:
		IF st_config.b_config_fertig THEN
			fb_state_entry.i16_next_step := INIT;
		END_IF

(*=======================================================*)
	INIT:
		IF fb_state_entry.E THEN
			fb_ton_wz.IN := FALSE;
			fb_ton_uez.IN := FALSE;
			fb_ton_quitt.IN := FALSE;
			st_ctrl_out.b_fehler := FALSE;
			st_ctrl_out.b_bereit := FALSE;
			st_ctrl_out.b_fertig := FALSE;
			zyl_bandfaenger.st_ctrl.in.b_ausfahren := FALSE;
			zyl_bandfaenger.st_ctrl.in.b_einfahren := FALSE;
			 zyl_bandklemmen.st_ctrl.in.b_ausfahren := FALSE;
			 zyl_bandklemmen.st_ctrl.in.b_einfahren := FALSE;
			sm_fehler_bandvorschub := FALSE;
			sm_keine_busverbindung := FALSE;
		END_IF

		(*-----------------------Weiterschaltbedingungen----------------------------*)
		IF st_ctrl_in.b_init THEN
			zyl_bandfaenger.st_ctrl.in.b_quittieren := FALSE;
			 zyl_bandklemmen.st_ctrl.in.b_quittieren := FALSE;
			IF gst_datensatz.st_md.b_wt_transport_simulation THEN
				fb_state_entry.i16_next_step := BEREIT;
			ELSE
				(*fb_state_entry.i16_next_step := 20; Bei nächster TSM-Änderung bitte aktivieren*)
				fb_state_entry.i16_next_step := BEREIT;
			END_IF
		END_IF

(*=======================================================*)
	20: (* Prüfe, ob Busverbindung vorhanden ist *)

		(*-----------------------Weiterschaltbedingungen----------------------------*)
		IF e_wc_state THEN	(* Prüfe Busverbindung ( 0=Data valid, 1=Data invalid )*)
			sm_keine_busverbindung := TRUE;
			fb_state_entry.i16_next_step := FEHLER;
		ELSE
			fb_state_entry.i16_next_step := BEREIT;
		END_IF

(*=======================================================*)
	BEREIT:
		IF fb_state_entry.E THEN
			st_ctrl_out.b_bereit := TRUE;
		END_IF

		(*-----------------------Weiterschaltbedingungen----------------------------*)
		CASE gst_datensatz.st_wkz.i16_typ_bandeinzug OF
			BANDWECHSLER_V2:
				(* Versuchsablauf zum mehrfach Biegen eines Bandes *)
				(* Die Anzahl der Werkzeughübe zum Biegen wird durch das Bestückprogramm bestimmt *)
				IF b_einzug_stop AND nockenschaltwerk_bestueckachse.fb.arr_spur[SP_OT] THEN
					fb_state_entry.i16_next_step := 500;
				ELSE
					fb_state_entry.i16_next_step := 200;
				END_IF
			SERVO:
				;
		END_CASE;

(*===========================Bandvorschub mit GLS-Kontrolle============================*)
	200:	(* Warte auf Vorschubnocke  und Freigabe von der Bestückachse *)
		(* Die Freigabe erfolgt nur im normalen Produktionsablauf; nicht bei Bandwechsel, Einfädeln, ... da hier keine Überwachung erfolgen soll. *)

		(*-----------------------Weiterschaltbedingungen----------------------------*)
		IF fb_r_trig_nocke_einzug.Q AND gi16_betriebsart <> HAND AND st_ctrl_in.b_freigabe THEN
			b_hm_pos_flanke_vorschub := FALSE;
			b_hm_neg_flanke_vorschub := FALSE;
			fb_state_entry.i16_next_step := 210;
		END_IF

(*=======================================================*)
	210:	(* Band wird vorgeschoben *)
		(* Vorschubkontrolle durch positive Flanke *)
		IF fb_r_trig_vorschubkontrolle.Q THEN
			b_hm_pos_flanke_vorschub := TRUE;
		END_IF
		(* Vorschubkontrolle durch negative Flanke *)
		IF fb_f_trig_vorschubkontrolle.Q THEN
			b_hm_neg_flanke_vorschub := TRUE;
		END_IF

		(* bei abgeschalteten Nocken *)
		IF	NOT gst_datensatz.st_wkz.nockenschaltwerk_bestueckachse.arr_nocken[NO_PNEUMATIKBANDEINZUG_GLS].b_camvalid THEN
			b_hm_neg_flanke_vorschub := TRUE;
			b_hm_pos_flanke_vorschub := TRUE;
		END_IF
		(*-----------------------Weiterschaltbedingungen----------------------------*)
		IF fb_f_trig_nocke_einzug.Q THEN
			IF b_hm_pos_flanke_vorschub AND b_hm_neg_flanke_vorschub THEN
				fb_state_entry.i16_next_step := 200;
			ELSE
				sm_fehler_bandvorschub := TRUE;
				fb_state_entry.i16_next_step := FEHLER;
			END_IF
		ELSIF gi16_betriebsart = HAND OR NOT st_ctrl_in.b_freigabe THEN
			fb_state_entry.i16_next_step := 200;
		END_IF

(*=======================================================*)
	500:	(* Nocken deaktivieren und Bandfänger deaktivieren/einfahren sowie Bandklemmen ausfahren*)
		IF fb_state_entry.E THEN
			CASE gst_datensatz.st_wkz.i16_typ_bandeinzug OF

				BANDWECHSLER_V2:
					(* Bandwechsler V2 ohne Sensoren und anderen Zylindern *)
					gst_datensatz.st_wkz.nockenschaltwerk_bestueckachse.arr_nocken[NO_BW_BANDFAENGER_BAWEV2_EINFAHREN].b_camvalid := FALSE;
					gst_datensatz.st_wkz.nockenschaltwerk_bestueckachse.arr_nocken[NO_BW_BANDFAENGER_BAWEV2_AUSFAHREN].b_camvalid := FALSE;
					gst_datensatz.st_wkz.nockenschaltwerk_bestueckachse.arr_nocken[NO_BW_BANDKLEMMEN_BAWEV2_EINFAHREN].b_camvalid := FALSE;
					gst_datensatz.st_wkz.nockenschaltwerk_bestueckachse.arr_nocken[NO_BW_BANDKLEMMEN_BAWEV2_AUSFAHREN].b_camvalid := FALSE;
				SERVO:
					;
			END_CASE;

			zyl_bandfaenger.fb.b_no_gesteuert_im_norm_betrieb := TRUE;
			zyl_bandklemmen.fb.b_no_gesteuert_im_norm_betrieb := TRUE;
			(* Zylinder einfahren *)
			zyl_bandfaenger.st_ctrl.in.b_einfahren := TRUE;
			zyl_bandklemmen.st_ctrl.in.b_ausfahren := TRUE;
		END_IF

		(*-----------------------Weiterschaltbedingungen----------------------------*)
		IF zyl_bandfaenger.st_ctrl.out.b_eingefahren AND zyl_bandklemmen.st_ctrl.out.b_ausgefahren AND gb_ba_auto_kontroller THEN
			zyl_bandfaenger.st_ctrl.in.b_einfahren := FALSE;
			zyl_bandklemmen.st_ctrl.in.b_ausfahren := FALSE;
			fb_state_entry.i16_next_step := 510;
		END_IF

(*=======================================================*)
	510:
		IF fb_state_entry.E THEN
			;
		END_IF

		(*-----------------------Weiterschaltbedingungen----------------------------*)
		IF NOT b_einzug_stop THEN
			(* Bandwechsler V1 *)
			gst_datensatz.st_wkz.nockenschaltwerk_bestueckachse.arr_nocken[NO_BW_BANDFAENGER_EINFAHREN].b_camvalid := TRUE;
			gst_datensatz.st_wkz.nockenschaltwerk_bestueckachse.arr_nocken[NO_BW_BANDFAENGER_AUSFAHREN].b_camvalid := TRUE;
			gst_datensatz.st_wkz.nockenschaltwerk_bestueckachse.arr_nocken[NO_UW_BANDFAENGER_EINFAHREN].b_camvalid := TRUE;
			gst_datensatz.st_wkz.nockenschaltwerk_bestueckachse.arr_nocken[NO_UW_BANDFAENGER_AUSFAHREN].b_camvalid := TRUE;
			gst_datensatz.st_wkz.nockenschaltwerk_bestueckachse.arr_nocken[NO_BW_BANDKLEMMEN_EINFAHREN].b_camvalid := TRUE;
			gst_datensatz.st_wkz.nockenschaltwerk_bestueckachse.arr_nocken[NO_BW_BANDKLEMMEN_AUSFAHREN].b_camvalid := TRUE;
			gst_datensatz.st_wkz.nockenschaltwerk_bestueckachse.arr_nocken[NO_UW_BANDKLEMMEN_EINFAHREN].b_camvalid := TRUE;
			gst_datensatz.st_wkz.nockenschaltwerk_bestueckachse.arr_nocken[NO_UW_BANDKLEMMEN_AUSFAHREN].b_camvalid := TRUE;
			(* Bandwechsler V2 ohne Sensoren und anderen Zylindern *)
			gst_datensatz.st_wkz.nockenschaltwerk_bestueckachse.arr_nocken[NO_BW_BANDFAENGER_BAWEV2_EINFAHREN].b_camvalid := TRUE;
			gst_datensatz.st_wkz.nockenschaltwerk_bestueckachse.arr_nocken[NO_BW_BANDFAENGER_BAWEV2_AUSFAHREN].b_camvalid := TRUE;
			gst_datensatz.st_wkz.nockenschaltwerk_bestueckachse.arr_nocken[NO_BW_BANDKLEMMEN_BAWEV2_EINFAHREN].b_camvalid := TRUE;
			gst_datensatz.st_wkz.nockenschaltwerk_bestueckachse.arr_nocken[NO_BW_BANDKLEMMEN_BAWEV2_AUSFAHREN].b_camvalid := TRUE;

			zyl_bandfaenger.fb.b_no_gesteuert_im_norm_betrieb := FALSE;
			zyl_bandklemmen.fb.b_no_gesteuert_im_norm_betrieb := FALSE;
			fb_state_entry.i16_next_step := BEREIT;
		END_IF

(*=======================================================*)
	FEHLER:
		IF fb_state_entry.E THEN
			st_ctrl_out.b_fehler := TRUE;
			fb_ton_quitt.IN := FALSE;
			zyl_bandfaenger.st_ctrl.in.b_quittieren := FALSE;
			zyl_bandklemmen.st_ctrl.in.b_quittieren := FALSE;
		END_IF

		(*-----------------------Weiterschaltbedingungen----------------------------*)
		IF st_ctrl_in.b_quitt AND NOT fb_state_entry.E THEN
			st_ctrl_out.b_fehler := FALSE;
			zyl_bandfaenger.st_ctrl.in.b_quittieren := TRUE;
			zyl_bandklemmen.st_ctrl.in.b_quittieren := TRUE;
			fb_ton_quitt.IN := TRUE;
		END_IF

		IF fb_ton_quitt.Q THEN
			fb_ton_quitt.IN := FALSE;
			fb_state_entry.i16_next_step := INIT;
		END_IF

(*=======================================================*)
	STOP:
		IF fb_state_entry.E THEN
			fb_ton_quitt.IN := FALSE;
			zyl_bandfaenger.st_ctrl.in.b_quittieren := FALSE;
			zyl_bandklemmen.st_ctrl.in.b_quittieren := FALSE;
		END_IF

		(*-----------------------Weiterschaltbedingungen----------------------------*)
		IF st_ctrl_in.b_quitt AND NOT fb_state_entry.E THEN
			fb_ton_quitt.IN := TRUE;
			zyl_bandfaenger.st_ctrl.in.b_quittieren := TRUE;
			zyl_bandklemmen.st_ctrl.in.b_quittieren := TRUE;
		END_IF

		IF fb_ton_quitt.Q THEN
			fb_ton_quitt.IN := FALSE;
			fb_state_entry.i16_next_step := INIT;
		END_IF
END_CASE

fb_state_entry(
	i16_next_step:= , 
	i16_pos:= 2,
	s_debugtext:= ,
	E=> , 
	X=> , 
	i16_step=> ,
	i16_last_step=> );

IF st_config.b_config_fertig THEN
	(* Fehlermeldungen und Betriebsmeldungen ab dem Startindex in die globalen Meldungsarrays schreiben *)
	garr_stoermeldungen[st_config.i16_meld_startindex + 0] := sm_fehler_bandvorschub;
	garr_stoermeldungen[st_config.i16_meld_startindex + 1] := FALSE;(* belegt  durch Bandeinzugskontroller 1720 *)
	garr_stoermeldungen[st_config.i16_meld_startindex + 2] := FALSE;(* belegt  durch Bandeinzugskontroller 1720 *)
	garr_stoermeldungen[st_config.i16_meld_startindex + 3] := sm_keine_busverbindung;
	garr_stoermeldungen[st_config.i16_meld_startindex + 4] := FALSE;
	garr_stoermeldungen[st_config.i16_meld_startindex + 5] := FALSE;
	garr_stoermeldungen[st_config.i16_meld_startindex + 6] := FALSE;
	garr_stoermeldungen[st_config.i16_meld_startindex + 7] := FALSE;
	garr_stoermeldungen[st_config.i16_meld_startindex + 8] := FALSE;
	garr_stoermeldungen[st_config.i16_meld_startindex + 9] := FALSE;
	garr_stoermeldungen[st_config.i16_meld_startindex + 10] := FALSE;
	garr_stoermeldungen[st_config.i16_meld_startindex + 11] := FALSE;
	garr_stoermeldungen[st_config.i16_meld_startindex + 12] := FALSE;
	garr_stoermeldungen[st_config.i16_meld_startindex + 13] := FALSE;
	garr_stoermeldungen[st_config.i16_meld_startindex + 14] := FALSE;
	garr_stoermeldungen[st_config.i16_meld_startindex + 15] := FALSE;
	garr_stoermeldungen[st_config.i16_meld_startindex + 16] := FALSE;
	garr_stoermeldungen[st_config.i16_meld_startindex + 17] := FALSE;
	garr_stoermeldungen[st_config.i16_meld_startindex + 18] := FALSE;
	garr_stoermeldungen[st_config.i16_meld_startindex + 19] := FALSE;
	
	garr_betriebsmeldungen[st_config.i16_meld_startindex + 0] := FALSE;
	garr_betriebsmeldungen[st_config.i16_meld_startindex + 1] := FALSE;
	garr_betriebsmeldungen[st_config.i16_meld_startindex + 2] := FALSE;
	garr_betriebsmeldungen[st_config.i16_meld_startindex + 3] := FALSE;
	garr_betriebsmeldungen[st_config.i16_meld_startindex + 4] := FALSE;
	garr_betriebsmeldungen[st_config.i16_meld_startindex + 5] := FALSE;
	garr_betriebsmeldungen[st_config.i16_meld_startindex + 6] := FALSE;
	garr_betriebsmeldungen[st_config.i16_meld_startindex + 7] := FALSE;
	garr_betriebsmeldungen[st_config.i16_meld_startindex + 8] := FALSE;
	garr_betriebsmeldungen[st_config.i16_meld_startindex + 9] := FALSE;
	garr_betriebsmeldungen[st_config.i16_meld_startindex + 10] := FALSE;
	garr_betriebsmeldungen[st_config.i16_meld_startindex + 11] := FALSE;
	garr_betriebsmeldungen[st_config.i16_meld_startindex + 12] := FALSE;
	garr_betriebsmeldungen[st_config.i16_meld_startindex + 13] := FALSE;
	garr_betriebsmeldungen[st_config.i16_meld_startindex + 14] := FALSE;
	garr_betriebsmeldungen[st_config.i16_meld_startindex + 15] := FALSE;
	garr_betriebsmeldungen[st_config.i16_meld_startindex + 16] := FALSE;
	garr_betriebsmeldungen[st_config.i16_meld_startindex + 17] := FALSE;
	garr_betriebsmeldungen[st_config.i16_meld_startindex + 18] := FALSE;
	garr_betriebsmeldungen[st_config.i16_meld_startindex + 19] := FALSE;
END_IF
END_PROGRAM

(* POU Maschine1720/ST_Bandeinzug_Kontroller_1720, ST *)
PROGRAM ST_Bandeinzug_Kontroller_1720
VAR_INPUT
	st_config							: struct_config;
	st_ctrl_in							: struct_ctrl_in;
END_VAR
VAR_IN_OUT
	st_visu							: struct_visu;
END_VAR
VAR_OUTPUT
	st_ctrl_out						: struct_ctrl_out;
END_VAR
VAR
	fb_ton_wz						: TON;
	fb_ton_uez						: TON;
	fb_ton_quitt						: TON;
	fb_state_entry						: ST_StateEntry;
	e_ls_bandende_re				AT %I* : BOOL;
	e_ls_bandende_li					AT %I* : BOOL;

	fb_r_trig_vorschubkontrolle_li		: R_TRIG;
	fb_f_trig_vorschubkontrolle_li		: F_TRIG;
	fb_r_trig_nocke_einzug				: R_TRIG;
	fb_f_trig_nocke_einzug				: F_TRIG;
	b_hm_pos_flanke_vorschub_li		: BOOL := FALSE;
	b_hm_neg_flanke_vorschub_li		: BOOL := FALSE;
	sm_fehler_bandvorschub_li			: BOOL := FALSE;
	fb_r_trig_vorschubkontrolle_re		: R_TRIG;
	fb_f_trig_vorschubkontrolle_re		: F_TRIG;
	b_hm_pos_flanke_vorschub_re		: BOOL := FALSE;
	b_hm_neg_flanke_vorschub_re		: BOOL := FALSE;
	sm_fehler_bandvorschub_re			: BOOL := FALSE;
	sm_keine_busverbindung			: BOOL := FALSE;

	e_wc_state							AT %I* : BOOL;	(* 0=Data valid, 1=Data invalid *)
	e_gls_bandvorschubkontrolle_li		AT %I* : BOOL;
	e_gls_bandvorschubkontrolle_re		AT %I* : BOOL;
END_VAR
(* Zeiten *)
fb_ton_wz(IN:= , PT:= , Q=>  , ET=> );
fb_ton_uez(IN:= , PT:= , Q=>  , ET=> );
fb_ton_quitt(IN:= , PT:= t#100ms, Q=> , ET=> );

(* Flanken *)
fb_f_trig_vorschubkontrolle_li(CLK:= e_gls_bandvorschubkontrolle_li, Q=> );
fb_r_trig_vorschubkontrolle_li(CLK:= e_gls_bandvorschubkontrolle_li, Q=> );
fb_f_trig_nocke_einzug(CLK:= nockenschaltwerk_bestueckachse.fb.arr_spur[SP_PNEUMATIKBANDEINZUG_GLS], Q=> );
fb_r_trig_nocke_einzug(CLK:= nockenschaltwerk_bestueckachse.fb.arr_spur[SP_PNEUMATIKBANDEINZUG_GLS], Q=> );
fb_f_trig_vorschubkontrolle_re(CLK:= e_gls_bandvorschubkontrolle_re, Q=> );
fb_r_trig_vorschubkontrolle_re(CLK:= e_gls_bandvorschubkontrolle_re, Q=> );

(*neue Haltezylinder für Bandklemmeinzug*)
(*bei Steuerung Ein oben bei Steuerung Aus wird selbständig über Federkraft geklemmt*)
IF ST_Safetyprogramm.se_steuerung_ein THEN
	zyl_bawe_halter_li.st_ctrl.in.b_einfahren := TRUE;
	zyl_bawe_halter_re.st_ctrl.in.b_einfahren := TRUE;
END_IF

(* Toplevel *)
IF fb_state_entry.i16_next_step > INIT AND fb_state_entry.i16_next_step < FEHLER THEN
	IF fb_state_entry.i16_next_step < STOP THEN
		IF st_ctrl_in.b_stop THEN
			fb_state_entry.i16_next_step := STOP;
		END_IF
	END_IF
	(* Allgemeine Fehler *)
	IF	NOT gst_datensatz.st_md.b_wt_transport_simulation AND
		(zyl_bandfaenger_li.st_ctrl.out.b_fehler OR
		zyl_bandklemmen_li.st_ctrl.out.b_fehler OR
		zyl_bandfaenger_re.st_ctrl.out.b_fehler OR
		zyl_bandklemmen_re.st_ctrl.out.b_fehler OR
		zyl_bawe_halter_li.st_ctrl.out.b_fehler OR
		zyl_bawe_halter_re.st_ctrl.out.b_fehler)
		THEN
			fb_state_entry.i16_next_step := FEHLER;
	(* Zylinder im Handbetrieb *)
	ELSIF	 gi16_betriebsart = HAND AND (
			(st_visu.st_zyl.i16_nr_zyl_im_handbetrieb = zyl_bandfaenger_li.fb.st_config.i16_identnummer OR
			st_visu.st_zyl.i16_nr_zyl_im_handbetrieb = zyl_bandfaenger_li.fb.st_config.i16_identnummer OR
			st_visu.st_zyl.i16_nr_zyl_im_handbetrieb = zyl_bandfaenger_re.fb.st_config.i16_identnummer OR
			st_visu.st_zyl.i16_nr_zyl_im_handbetrieb = zyl_bandklemmen_re.fb.st_config.i16_identnummer OR
			st_visu.st_zyl.i16_nr_zyl_im_handbetrieb = zyl_bawe_halter_li.fb.st_config.i16_identnummer OR
			st_visu.st_zyl.i16_nr_zyl_im_handbetrieb = zyl_bawe_halter_re.fb.st_config.i16_identnummer))
			THEN
				fb_state_entry.i16_next_step := FEHLER;
	END_IF
END_IF

(* ======================================Schrittkette======================================== *)
fb_state_entry(
	i16_next_step:= ,
	i16_pos:= 1,
	s_debugtext:= ,
	E=> ,
	X=> , 
	i16_step=> ,
	i16_last_step=> );

CASE fb_state_entry.i16_step OF
(*=======================================================*)
	INIT_OBJ:
		IF st_config.b_config_fertig THEN
			fb_state_entry.i16_next_step := INIT;
		END_IF

(*=======================================================*)
	INIT:
		IF fb_state_entry.E THEN
			fb_ton_wz.IN := FALSE;
			fb_ton_uez.IN := FALSE;
			fb_ton_quitt.IN := FALSE;
			st_ctrl_out.b_fehler := FALSE;
			st_ctrl_out.b_bereit := FALSE;
			st_ctrl_out.b_fertig := FALSE;
			zyl_bandfaenger_li.st_ctrl.in.b_ausfahren := FALSE;
			zyl_bandfaenger_li.st_ctrl.in.b_einfahren := FALSE;
			 zyl_bandklemmen_li.st_ctrl.in.b_ausfahren := FALSE;
			 zyl_bandklemmen_li.st_ctrl.in.b_einfahren := FALSE;
			zyl_bandfaenger_re.st_ctrl.in.b_ausfahren := FALSE;
			zyl_bandfaenger_re.st_ctrl.in.b_einfahren := FALSE;
			 zyl_bandklemmen_re.st_ctrl.in.b_ausfahren := FALSE;
			 zyl_bandklemmen_re.st_ctrl.in.b_einfahren := FALSE;
			sm_fehler_bandvorschub_li := FALSE;
			sm_fehler_bandvorschub_re := FALSE;
			sm_keine_busverbindung := FALSE;
		END_IF

		(*-----------------------Weiterschaltbedingungen----------------------------*)
		IF st_ctrl_in.b_init THEN
			zyl_bandfaenger_li.st_ctrl.in.b_quittieren := FALSE;
			zyl_bandklemmen_li.st_ctrl.in.b_quittieren := FALSE;
			zyl_bandfaenger_re.st_ctrl.in.b_quittieren := FALSE;
			zyl_bandklemmen_re.st_ctrl.in.b_quittieren := FALSE;
			zyl_bawe_halter_li.st_ctrl.in.b_quittieren := FALSE;
			zyl_bawe_halter_re.st_ctrl.in.b_quittieren := FALSE;
			IF gst_datensatz.st_md.b_wt_transport_simulation THEN
				fb_state_entry.i16_next_step := BEREIT;
			ELSE
				(*fb_state_entry.i16_next_step := 20; Bei nächster TSM-Änderung bitte aktivieren*)
				fb_state_entry.i16_next_step := BEREIT;
			END_IF
		END_IF

(*=======================================================*)
	20: (* Prüfe, ob Busverbindung vorhanden ist *)

		(*-----------------------Weiterschaltbedingungen----------------------------*)
		IF e_wc_state THEN	(* Prüfe Busverbindung ( 0=Data valid, 1=Data invalid )*)
			sm_keine_busverbindung := TRUE;
			fb_state_entry.i16_next_step := FEHLER;
		ELSE
			fb_state_entry.i16_next_step := BEREIT;
		END_IF

(*=======================================================*)
	BEREIT:
		IF fb_state_entry.E THEN
			st_ctrl_out.b_bereit := TRUE;
		END_IF

		(*-----------------------Weiterschaltbedingungen----------------------------*)
		CASE gst_datensatz.st_wkz.i16_typ_bandeinzug OF

			STANDARD_2FACH_V2:
				fb_state_entry.i16_next_step := 200;


			BANDWECHSLER_V2:
				(* Den Bandwechsler gibt es nur bei BSH1700 *)
				;
		END_CASE;

(*===========================Bandvorschub mit GLS-Kontrolle============================*)
	200:	(* Warte auf Vorschubnocke  und Freigabe von der Bestückachse *)
		(* Die Freigabe erfolgt nur im normalen Produktionsablauf; nicht bei Bandwechsel, Einfädeln, ... da hier keine Überwachung erfolgen soll. *)

		(*-----------------------Weiterschaltbedingungen----------------------------*)
		IF fb_r_trig_nocke_einzug.Q AND gi16_betriebsart <> HAND AND st_ctrl_in.b_freigabe THEN
			b_hm_pos_flanke_vorschub_li := FALSE;
			b_hm_neg_flanke_vorschub_li := FALSE;
			b_hm_pos_flanke_vorschub_re := FALSE;
			b_hm_neg_flanke_vorschub_re := FALSE;
			fb_state_entry.i16_next_step := 210;
		END_IF

(*=======================================================*)
	210:	(* Band links bzw. rechts wird vorgeschoben *)
		(* Vorschubkontrolle durch positive Flanke *)
		IF fb_r_trig_vorschubkontrolle_li.Q THEN
			b_hm_pos_flanke_vorschub_li := TRUE;
		END_IF
		IF fb_r_trig_vorschubkontrolle_re.Q THEN
			b_hm_pos_flanke_vorschub_re := TRUE;
		END_IF
		(* Vorschubkontrolle durch negative Flanke *)
		IF fb_f_trig_vorschubkontrolle_li.Q THEN
			b_hm_neg_flanke_vorschub_li := TRUE;
		END_IF
		IF fb_f_trig_vorschubkontrolle_re.Q THEN
			b_hm_neg_flanke_vorschub_re := TRUE;
		END_IF


		(*-----------------------Weiterschaltbedingungen----------------------------*)
		IF fb_f_trig_nocke_einzug.Q THEN
			IF 	b_hm_pos_flanke_vorschub_li AND b_hm_neg_flanke_vorschub_li AND
				b_hm_pos_flanke_vorschub_re AND b_hm_neg_flanke_vorschub_re
				THEN
					fb_state_entry.i16_next_step := 200;
			ELSE
				IF NOT b_hm_pos_flanke_vorschub_li OR NOT b_hm_neg_flanke_vorschub_li THEN
					sm_fehler_bandvorschub_li := TRUE;
				END_IF
				IF NOT b_hm_pos_flanke_vorschub_re OR NOT b_hm_neg_flanke_vorschub_re THEN
					sm_fehler_bandvorschub_re := TRUE;
				END_IF
				fb_state_entry.i16_next_step := FEHLER;
			END_IF
		ELSIF gi16_betriebsart = HAND THEN
			fb_state_entry.i16_next_step := 200;
		END_IF

(*=======================================================*)
	FEHLER:
		IF fb_state_entry.E THEN
			st_ctrl_out.b_fehler := TRUE;
			fb_ton_quitt.IN := FALSE;
			zyl_bandfaenger_li.st_ctrl.in.b_quittieren := FALSE;
			zyl_bandklemmen_li.st_ctrl.in.b_quittieren := FALSE;
			zyl_bandfaenger_re.st_ctrl.in.b_quittieren := FALSE;
			zyl_bandklemmen_re.st_ctrl.in.b_quittieren := FALSE;
			zyl_bawe_halter_li.st_ctrl.in.b_quittieren := FALSE;
			zyl_bawe_halter_re.st_ctrl.in.b_quittieren := FALSE;
		END_IF

		(*-----------------------Weiterschaltbedingungen----------------------------*)
		IF st_ctrl_in.b_quitt AND NOT fb_state_entry.E THEN
			st_ctrl_out.b_fehler := FALSE;
			zyl_bandfaenger_li.st_ctrl.in.b_quittieren := TRUE;
			zyl_bandklemmen_li.st_ctrl.in.b_quittieren := TRUE;
			zyl_bandfaenger_re.st_ctrl.in.b_quittieren := TRUE;
			zyl_bandklemmen_re.st_ctrl.in.b_quittieren := TRUE;
			zyl_bawe_halter_li.st_ctrl.in.b_quittieren := TRUE;
			zyl_bawe_halter_re.st_ctrl.in.b_quittieren := TRUE;
			fb_ton_quitt.IN := TRUE;
		END_IF

		IF fb_ton_quitt.Q THEN
			fb_ton_quitt.IN := FALSE;
			fb_state_entry.i16_next_step := INIT;
		END_IF

(*=======================================================*)
	STOP:
		IF fb_state_entry.E THEN
			fb_ton_quitt.IN := FALSE;
			zyl_bandfaenger_li.st_ctrl.in.b_quittieren := FALSE;
			zyl_bandklemmen_li.st_ctrl.in.b_quittieren := FALSE;
			zyl_bandfaenger_re.st_ctrl.in.b_quittieren := FALSE;
			zyl_bandklemmen_re.st_ctrl.in.b_quittieren := FALSE;
			zyl_bawe_halter_li.st_ctrl.in.b_quittieren := FALSE;
			zyl_bawe_halter_re.st_ctrl.in.b_quittieren := FALSE;
		END_IF

		(*-----------------------Weiterschaltbedingungen----------------------------*)
		IF st_ctrl_in.b_quitt AND NOT fb_state_entry.E THEN
			fb_ton_quitt.IN := TRUE;
			zyl_bandfaenger_li.st_ctrl.in.b_quittieren := TRUE;
			zyl_bandklemmen_li.st_ctrl.in.b_quittieren := TRUE;
			zyl_bandfaenger_re.st_ctrl.in.b_quittieren := TRUE;
			zyl_bandklemmen_re.st_ctrl.in.b_quittieren := TRUE;
			zyl_bawe_halter_li.st_ctrl.in.b_quittieren := TRUE;
			zyl_bawe_halter_re.st_ctrl.in.b_quittieren := TRUE;
		END_IF

		IF fb_ton_quitt.Q THEN
			fb_ton_quitt.IN := FALSE;
			fb_state_entry.i16_next_step := INIT;
		END_IF
END_CASE

fb_state_entry(
	i16_next_step:= , 
	i16_pos:= 2,
	s_debugtext:= ,
	E=> , 
	X=> , 
	i16_step=> ,
	i16_last_step=> );

IF st_config.b_config_fertig THEN
	(* Fehlermeldungen und Betriebsmeldungen ab dem Startindex in die globalen Meldungsarrays schreiben *)
	garr_stoermeldungen[st_config.i16_meld_startindex + 0] := FALSE;(* belegt  durch Bandeinzugskontroller 1700 *)
	garr_stoermeldungen[st_config.i16_meld_startindex + 1] := sm_fehler_bandvorschub_li;
	garr_stoermeldungen[st_config.i16_meld_startindex + 2] := sm_fehler_bandvorschub_re;
	garr_stoermeldungen[st_config.i16_meld_startindex + 3] := sm_keine_busverbindung;
	garr_stoermeldungen[st_config.i16_meld_startindex + 4] := FALSE;
	garr_stoermeldungen[st_config.i16_meld_startindex + 5] := FALSE;
	garr_stoermeldungen[st_config.i16_meld_startindex + 6] := FALSE;
	garr_stoermeldungen[st_config.i16_meld_startindex + 7] := FALSE;
	garr_stoermeldungen[st_config.i16_meld_startindex + 8] := FALSE;
	garr_stoermeldungen[st_config.i16_meld_startindex + 9] := FALSE;
	garr_stoermeldungen[st_config.i16_meld_startindex + 10] := FALSE;
	garr_stoermeldungen[st_config.i16_meld_startindex + 11] := FALSE;
	garr_stoermeldungen[st_config.i16_meld_startindex + 12] := FALSE;
	garr_stoermeldungen[st_config.i16_meld_startindex + 13] := FALSE;
	garr_stoermeldungen[st_config.i16_meld_startindex + 14] := FALSE;
	garr_stoermeldungen[st_config.i16_meld_startindex + 15] := FALSE;
	garr_stoermeldungen[st_config.i16_meld_startindex + 16] := FALSE;
	garr_stoermeldungen[st_config.i16_meld_startindex + 17] := FALSE;
	garr_stoermeldungen[st_config.i16_meld_startindex + 18] := FALSE;
	garr_stoermeldungen[st_config.i16_meld_startindex + 19] := FALSE;
	
	garr_betriebsmeldungen[st_config.i16_meld_startindex + 0] := FALSE;
	garr_betriebsmeldungen[st_config.i16_meld_startindex + 1] := FALSE;
	garr_betriebsmeldungen[st_config.i16_meld_startindex + 2] := FALSE;
	garr_betriebsmeldungen[st_config.i16_meld_startindex + 3] := FALSE;
	garr_betriebsmeldungen[st_config.i16_meld_startindex + 4] := FALSE;
	garr_betriebsmeldungen[st_config.i16_meld_startindex + 5] := FALSE;
	garr_betriebsmeldungen[st_config.i16_meld_startindex + 6] := FALSE;
	garr_betriebsmeldungen[st_config.i16_meld_startindex + 7] := FALSE;
	garr_betriebsmeldungen[st_config.i16_meld_startindex + 8] := FALSE;
	garr_betriebsmeldungen[st_config.i16_meld_startindex + 9] := FALSE;
	garr_betriebsmeldungen[st_config.i16_meld_startindex + 10] := FALSE;
	garr_betriebsmeldungen[st_config.i16_meld_startindex + 11] := FALSE;
	garr_betriebsmeldungen[st_config.i16_meld_startindex + 12] := FALSE;
	garr_betriebsmeldungen[st_config.i16_meld_startindex + 13] := FALSE;
	garr_betriebsmeldungen[st_config.i16_meld_startindex + 14] := FALSE;
	garr_betriebsmeldungen[st_config.i16_meld_startindex + 15] := FALSE;
	garr_betriebsmeldungen[st_config.i16_meld_startindex + 16] := FALSE;
	garr_betriebsmeldungen[st_config.i16_meld_startindex + 17] := FALSE;
	garr_betriebsmeldungen[st_config.i16_meld_startindex + 18] := FALSE;
	garr_betriebsmeldungen[st_config.i16_meld_startindex + 19] := FALSE;
END_IF
END_PROGRAM

(* POU MAINs/MAIN_STANDARD, ST *)
PROGRAM MAIN_STANDARD
VAR
END_VAR
CASE gst_datensatz.st_md.i16_typ_zelle OF
	KEINE_ZELLE:
		;
	BESTUECKZELLE_1700:
		IF visu.s_akt_sprache <> 'en' THEN
			ST_AutoCheckIn( i_IntervalDay:=7 );
		END_IF
		ST_SaveAndLoad();
		ST_Datainit_Stationen();
		ST_Datainit_Achsen();

		ST_EthercatDiag();

		(* Grundmaschine *)
		EtherCatDiag[1]( );
		EtherCatDiag[1].st_config.b_station_aktiv := TRUE;

		(* Hublift links *)
		EtherCatDiag[2]( );
		EtherCatDiag[2].st_config.b_station_aktiv := gst_datensatz.st_md.b_hublift_links_aktiv;

		(* Hublift rechts *)
		EtherCatDiag[3]( );
		EtherCatDiag[3].st_config.b_station_aktiv := gst_datensatz.st_md.b_hublift_rechts_aktiv;

		(* Bandeinzug *)
		(* Bandeinzug nicht aufrufen, weil in allen TSM der Mulitpol A170 für die Rasterfolie drin ist und dieser
		in keinem normalen Bandeinzug
		Bei normalem Bandeinzug kommt immer Fehler Busverbindung *)
		(*EtherCatDiag[4]( );
		EtherCatDiag[4].st_config.b_station_aktiv := NOT gst_datensatz.st_md.b_wt_transport_simulation;*)

		ST_UPS(st_config:= UPS.st_config,
			st_ctrl_in:= UPS.st_ctrl.in,
			b_Ups := TRUE,
			st_ctrl_out=> UPS.st_ctrl.out);

		ST_RoutingBackpanel(
			st_config:= routing_backpanel.st_config,
			st_ctrl_in:= routing_backpanel.st_ctrl.in,
			st_ctrl_out=> routing_backpanel.st_ctrl.out);

		ST_MotionFunctionPoints(
			st_ctrl_in:= edit_mfps.st_ctrl.in,
			st_ctrl_out=> edit_mfps.st_ctrl.out);

		ST_Schreibe_Persistente_Daten(
			bExecute:= ,
			bQuit:= ,
			t_schreibintervall:= t#60s,
			b_steuerung_ein:= ST_Safetyprogramm.se_steuerung_ein,
			bBusy=> ,
			bError=> ,
			nErrId=> );

		ST_System_DateAndTime();

		betriebsstundenzaehler.fb(
			b_eingekuppelt:= (ST_Z_Achse.fb_state_entry.i16_step > BEREIT AND ST_Z_Achse.fb_state_entry.i16_step < HALT) AND (gi16_betriebsart = AUTO),
			b_reset:= ,
			i32_betriebssekundenzaehler_in:= gst_datensatz.st_md.i32_betriebssekundenzaehler,
			i32_betriebssekundenzaehler=> gst_datensatz.st_md.i32_betriebssekundenzaehler);

		ST_Tuerverriegelung(
			e_quittiertaste:= ST_Safetyprogramm.se_quittiertaste);

		ST_LampeMaterialMangel(b_materialmangel:=  );

		ST_Zylinder();

		ST_start_OSK(bExecute:= ST_Safetyprogramm.se_quittiertaste);

		ST_Euchner_Handbedienpult();

		ST_TippTasten(
			i16_akt_stufe:= ,
			b_initialisierungsphase:= ,
			b_einfaedeln_aktiv:= ,
			st_visu:= visu,
			st_visu_hinten:= visu_hinten);

		ST_Betriebsarten(st_config:= betriebsarten.st_config);

		(* Übernahme der Daten aus der Datenbank: Beladen und Abgabe greifen dann auf diese Konfiguration zu *)
		wt_transport_kontroller.st_config.b_station_aktiv := gst_datensatz.st_md.b_wt_transport_aktiv;
		wt_transport_kontroller.st_config.b_station_in_simulation := gst_datensatz.st_md.b_wt_transport_simulation;

		ST_WT_Transport_Kontroller(
			st_config:= wt_transport_kontroller.st_config,
			st_ctrl_in:= wt_transport_kontroller.st_ctrl.in,
			st_visu:= visu,
			st_ctrl_out=> wt_transport_kontroller.st_ctrl.out);

		(* Aktivierung durch den Kontroller *)
		wt_transport_abgabe.st_config.b_station_aktiv := gst_datensatz.st_md.b_wt_transport_aktiv;
		wt_transport_abgabe.st_config.b_station_in_simulation := gst_datensatz.st_md.b_wt_transport_simulation;

		ST_WT_Transport_Abgabe(
			st_config:= wt_transport_abgabe.st_config,
			st_ctrl_in:= wt_transport_abgabe.st_ctrl.in,
			e_station_nachher_in_erlaubnis:= ,
			e_station_nachher_in_angekommen:= ,
			st_visu:= wt_transport_abgabe.st_visu,
			st_ctrl_out=> wt_transport_abgabe.st_ctrl.out,
			a_station_nachher_out_anforderung=> a_smema_station_nachher_out_anforderung,
			a_station_nachher_out_abgegeben=> a_smema_station_nachher_out_abgegeben);

		hublift_rechts.st_config.b_station_aktiv := gst_datensatz.st_md.b_hublift_rechts_aktiv;
		hublift_rechts.st_config.b_station_in_simulation := gst_datensatz.st_md.b_hublift_rechts_simulation;

		ST_Hublift_rechts(
			st_config:= hublift_rechts.st_config,
			st_ctrl_in:= hublift_rechts.st_ctrl.in,
			e_station_vorher_in_anforderung	:= ,
			e_station_vorher_in_abgegeben:= ,
			st_visu:= hublift_rechts.st_visu,
			st_ctrl_out=> hublift_rechts.st_ctrl.out,
			a_station_vorher_out_erlaubnis=> ,
			a_station_vorher_out_angekommen=> );
		IF hublift_rechts.st_config.b_station_aktiv OR hublift_rechts.st_config.b_station_in_simulation THEN
			ST_Hublift_rechts.e_station_vorher_in_abgegeben := ST_WT_Transport_Abgabe.a_station_nachher_out_abgegeben;
			ST_Hublift_rechts.e_station_vorher_in_anforderung := ST_WT_Transport_Abgabe.a_station_nachher_out_anforderung;
			ST_WT_Transport_Abgabe.e_station_nachher_in_angekommen := ST_Hublift_rechts.a_station_vorher_out_angekommen;
			ST_WT_Transport_Abgabe.e_station_nachher_in_erlaubnis := ST_Hublift_rechts.a_station_vorher_out_erlaubnis;
		ELSE
			ST_WT_Transport_Abgabe.e_station_nachher_in_angekommen := e_smema_station_nachher_in_angekommen;
			ST_WT_Transport_Abgabe.e_station_nachher_in_erlaubnis := e_smema_station_nachher_in_erlaubnis;
		END_IF

		balluff_tag_reader.fb(
			st_config:= balluff_tag_reader.fb.st_config,
			i16_addresse:= ,
			i16_anzahl_byte:= ,
			s_schreib_daten:= ,
			st_ctrl_in:= balluff_tag_reader.st_ctrl.in,
			s_lese_daten=> ,
			st_ctrl_out=> balluff_tag_reader.st_ctrl.out);

		barcode.fb(
			st_config:= barcode.fb.st_config,
			st_barcode_daten := gst_barcode_daten,
			b_steuerung_ein := ST_Safetyprogramm.se_steuerung_ein,
			b_bandende_links := ST_Bandwechsel_Kontroller.e_ls_bandende_li ,
			b_bandende_rechts := ST_Bandwechsel_Kontroller.e_ls_bandende_re,
			b_bandende_1720 := ST_Bandeinzug_Kontroller_1720.e_ls_bandende_li,
			b_band_nicht_gescannt=> ST_LampeMaterialMangel.b_materialmangel[5]);

		visu_hinten.in.bandfreigabe[0] := gst_barcode_daten.b_band_rechts_ok;
		visu_hinten.in.bandfreigabe[1] := gst_barcode_daten.b_band_links_ok;
		visu_hinten.in.band_ID[0] := gst_barcode_daten.b_band_ID_rechts_ok;
		visu_hinten.in.band_ID[1] := gst_barcode_daten.b_band_ID_links_ok;

		ST_VisuRouter();

		ST_Message_Produktion();

		ST_Bestueckachse(
			st_config_achse:= axis_bestueckachse.st_config,
			st_ctrl_in:= axis_bestueckachse.st_ctrl.in,
			e_steuerung_ein:= ST_Safetyprogramm.se_steuerung_ein,
			e_ba_mit_bedingungen:= ST_Safetyprogramm.se_ba_mit_bedingungen,
			e_tuere_vorne_offen:= ST_Safetyprogramm.se_tuere_vorne_offen,
			e_tuere_hinten_offen:= ST_Safetyprogramm.se_tuere_hinten_offen,
			st_visu:= axis_bestueckachse.st_visu,
			st_ctrl_out=> axis_bestueckachse.st_ctrl.out);

		ST_Z_Achse(
			st_config_achse:= axis_z_achse.st_config,
			st_ctrl_in:= axis_z_achse.st_ctrl.in,
			e_steuerung_ein:= ST_Safetyprogramm.se_steuerung_ein,
			e_ba_mit_bedingungen:= ST_Safetyprogramm.se_ba_mit_bedingungen,
			e_tuere_vorne_offen:= ST_Safetyprogramm.se_tuere_vorne_offen,
			e_tuere_hinten_offen:= ST_Safetyprogramm.se_tuere_hinten_offen,
			st_visu:= axis_z_achse.st_visu,
			st_ctrl_out=> axis_z_achse.st_ctrl.out,
			t_Z_Achse_ausfahren=>visu.ST_Service.t_Z_Achse_ausfahren,
			t_Bestueckung=>visu.ST_Service.t_Bestueckung,
			t_Z_Achse_einfahren=>visu.ST_Service.t_Z_Achse_einfahren);

		ST_TouchProbe();

		ST_Y_Achse(
			st_config_achse:= axis_y_achse.st_config,
			st_ctrl_in:= axis_y_achse.st_ctrl.in,
			e_steuerung_ein:= ST_Safetyprogramm.se_steuerung_ein,
			e_ba_mit_bedingungen:= ST_Safetyprogramm.se_ba_mit_bedingungen,
			e_tuere_vorne_offen:= ST_Safetyprogramm.se_tuere_vorne_offen,
			e_tuere_hinten_offen:= ST_Safetyprogramm.se_tuere_hinten_offen,
			e_not_steu_tuer_schutz_ok:= ,
			st_visu:= axis_y_achse.st_visu,
			st_ctrl_out=> axis_y_achse.st_ctrl.out);


		ST_Gesamthubzaehler();

		IF gst_Datensatz.st_md.b_anwahl_transport_achse THEN

			ST_WT_Transport_Achse(
				st_config_achse:= axis_transport_wt_achse.st_config,
				st_ctrl_in:= axis_transport_wt_achse.st_ctrl.in,
				e_steuerung_ein:= ST_Safetyprogramm.se_steuerung_ein,
				e_ba_mit_bedingungen:= ST_Safetyprogramm.se_ba_mit_bedingungen,
				e_tuere_vorne_offen:= ST_Safetyprogramm.se_tuere_vorne_offen,
				e_tuere_hinten_offen:= ST_Safetyprogramm.se_tuere_hinten_offen,
				st_visu:= axis_transport_wt_achse.st_visu,
				st_ctrl_out=> axis_transport_wt_achse.st_ctrl.out);

			wt_transport_warteposition_1700.st_config.b_station_aktiv := gst_datensatz.st_md.b_wt_transport_aktiv;
			wt_transport_warteposition_1700.st_config.b_station_in_simulation := gst_datensatz.st_md.b_wt_transport_simulation;

			ST_WT_Transport_Warteposition_1700(
				st_config:= wt_transport_warteposition_1700.st_config,
				st_ctrl_in:= wt_transport_warteposition_1700.st_ctrl.in,
				e_station_vorher_in_anforderung	:= ,
				e_station_vorher_in_abgegeben:= ,
				st_visu:= wt_transport_warteposition_1700.st_visu,
				st_ctrl_out=> wt_transport_warteposition_1700.st_ctrl.out,
				a_station_vorher_out_erlaubnis=> a_smema_station_vorher_out_erlaubnis,
				a_station_vorher_out_angekommen=> a_smema_station_vorher_out_angekommen);
	
			wt_transport_beladen_achse_1700.st_config.b_station_aktiv := gst_datensatz.st_md.b_wt_transport_aktiv;
			wt_transport_beladen_achse_1700.st_config.b_station_in_simulation := gst_datensatz.st_md.b_wt_transport_simulation;
	
			ST_WT_Transport_Beladen_Achse_1700(
				st_config:= wt_transport_beladen_achse_1700.st_config,
				st_ctrl_in:= wt_transport_beladen_achse_1700.st_ctrl.in,
				e_wt_im_aktionsfeld := balluff_tag_reader.fb.e_tag_im_aktionsfeld,
				st_visu:= wt_transport_beladen_achse_1700.st_visu,
				st_ctrl_out=> wt_transport_beladen_achse_1700.st_ctrl.out,
				t_WT_WechselZeit=>visu.ST_Service.t_WT_wechsel,
				t_traegerwechselzeit=>visu.ST_Service.t_traegerwechselzeit,
				t_Zentrierer_ausfahren=>visu.ST_Service.t_Zentrierer_ausfahren,
				t_Zentrierer_einfahren=>visu.ST_Service.t_Zentrierer_einfahren,
				t_komplett_zyklus=>visu.ST_Service.t_komplett_zyklus,);

		ELSE
			(* Aktivierung durch den Kontroller *)
			wt_transport_beladen.st_config.b_station_aktiv := gst_datensatz.st_md.b_wt_transport_aktiv;
			wt_transport_beladen.st_config.b_station_in_simulation := gst_datensatz.st_md.b_wt_transport_simulation;
	
			ST_WT_Transport_Beladen(
				st_config:= wt_transport_beladen.st_config,
				st_ctrl_in:= wt_transport_beladen.st_ctrl.in,
				e_station_vorher_in_anforderung	:= ,
				e_station_vorher_in_abgegeben:= ,
				st_visu:= wt_transport_beladen.st_visu,
				st_ctrl_out=> wt_transport_beladen.st_ctrl.out,
				a_station_vorher_out_erlaubnis=> a_smema_station_vorher_out_erlaubnis,
				a_station_vorher_out_angekommen=> a_smema_station_vorher_out_angekommen,
				t_WT_WechselZeit=>visu.ST_Service.t_WT_wechsel,
				t_traegerwechselzeit=>visu.ST_Service.t_traegerwechselzeit,
				t_Zentrierer_ausfahren=>visu.ST_Service.t_Zentrierer_ausfahren,
				t_Zentrierer_einfahren=>visu.ST_Service.t_Zentrierer_einfahren,
				t_komplett_zyklus=>visu.ST_Service.t_komplett_zyklus,);
		END_IF

		hublift_links.st_config.b_station_aktiv := gst_datensatz.st_md.b_hublift_links_aktiv;
		hublift_links.st_config.b_station_in_simulation := gst_datensatz.st_md.b_hublift_links_simulation;

		ST_Hublift_links(
			st_config:= hublift_links.st_config,
			st_ctrl_in:= hublift_links.st_ctrl.in,
			e_station_nachher_in_erlaubnis:= ,
			e_station_nachher_in_angekommen:= ,
			st_visu:= hublift_links.st_visu,
			st_ctrl_out=> hublift_links.st_ctrl.out,
			a_station_nachher_out_anforderung=> ,
			a_station_nachher_out_abgegeben=> );
		IF hublift_links.st_config.b_station_aktiv OR hublift_links.st_config.b_station_in_simulation THEN
			IF gst_Datensatz.st_md.b_anwahl_transport_achse THEN
				ST_WT_Transport_Warteposition_1700.e_station_vorher_in_abgegeben := ST_Hublift_links.a_station_nachher_out_abgegeben;
				ST_WT_Transport_Warteposition_1700.e_station_vorher_in_anforderung := ST_Hublift_links.a_station_nachher_out_anforderung;
				ST_Hublift_links.e_station_nachher_in_angekommen := ST_WT_Transport_Warteposition_1700.a_station_vorher_out_angekommen;
				ST_Hublift_links.e_station_nachher_in_erlaubnis := ST_WT_Transport_Warteposition_1700.a_station_vorher_out_erlaubnis;
			ELSE
				ST_WT_Transport_Beladen.e_station_vorher_in_abgegeben := ST_Hublift_links.a_station_nachher_out_abgegeben;
				ST_WT_Transport_Beladen.e_station_vorher_in_anforderung := ST_Hublift_links.a_station_nachher_out_anforderung;
				ST_Hublift_links.e_station_nachher_in_angekommen := ST_WT_Transport_Beladen.a_station_vorher_out_angekommen;
				ST_Hublift_links.e_station_nachher_in_erlaubnis := ST_WT_Transport_Beladen.a_station_vorher_out_erlaubnis;
			END_IF
		ELSE
			IF gst_Datensatz.st_md.b_anwahl_transport_achse THEN
				ST_WT_Transport_Warteposition_1700.e_station_vorher_in_abgegeben := e_smema_station_vorher_in_abgegeben;
				ST_WT_Transport_Warteposition_1700.e_station_vorher_in_anforderung := e_smema_station_vorher_in_anforderung;
			ELSE
				ST_WT_Transport_Beladen.e_station_vorher_in_abgegeben := e_smema_station_vorher_in_abgegeben;
				ST_WT_Transport_Beladen.e_station_vorher_in_anforderung := e_smema_station_vorher_in_anforderung;
			END_IF
		END_IF

		ST_Stoerungen_Quitt_1700(
			st_config:= stoerungen_quittieren.st_config,
			st_ctrl_in:= stoerungen_quittieren.st_ctrl.in,
			st_visu:= visu,
			st_visu_hinten:= visu_hinten,
			st_ctrl_out=> stoerungen_quittieren.st_ctrl.out,
			b_lampe_stoerung=> ST_Betriebsfreigaben.b_lampe_stoerung,
			b_lampe_produktion=> ST_Betriebsfreigaben.b_lampe_produktion);

		ST_Bandwechsel_Kontroller(
			st_config:= bandwechsel_kontroller.st_config,
			st_ctrl_in:= bandwechsel_kontroller.st_ctrl.in,
			st_visu:= visu,
			b_materialmangel=> ST_LampeMaterialMangel.b_materialmangel[3],
			st_ctrl_out=> bandwechsel_kontroller.st_ctrl.out);

		ST_Haspel_Kontroller_2H(
			t_abschaltzeit_motor:= haspel_kontroller.t_abschaltzeit_motor,
			b_drehrichtung_antrieb_links := gst_datensatz.st_wkz.b_laufrichtung_haspel_links,
			st_config:= haspel_kontroller.st_config,
			e_druckwaechter:= ST_Betriebsfreigaben.e_druckwaechter,
			e_steuerung_ein:= ST_Safetyprogramm.se_steuerung_ein,
			st_ctrl_in:= haspel_kontroller.st_ctrl.in,
			haspel1_ctrl_in:= haspel_li.st_ctrl.out,
			haspel2_ctrl_in:= haspel_re.st_ctrl.out,
			st_visu:= haspel_kontroller.st_visu,
			st_ctrl_out=> haspel_kontroller.st_ctrl.out,
			haspel1_ctrl_out=> haspel_li.st_ctrl.in,
			haspel2_ctrl_out=> haspel_re.st_ctrl.in,
			b_materialmangel_bandende=> ST_LampeMaterialMangel.b_materialmangel[0]);

		Haspel_Li.fb(
			t_wartezeit_bandende:= t#5s,
			b_bandende_Bandeinzug := ST_Bandwechsel_Kontroller.e_ls_bandende_li ,
			b_band_ok := gst_barcode_daten.b_band_links_ok AND gst_barcode_daten.b_band_ID_links_ok,
			st_config:= Haspel_Li.fb.st_config,
			st_ctrl_in:= Haspel_Li.st_ctrl.in,
			st_visu := Haspel_Li.st_visu,
			st_zyl_heben:= zyl_haspel_li_heben,
			st_zyl_abspulen:= zyl_haspel_li_abspulen,
			st_zyl_sperren:= zyl_haspel_li_sperren,
			st_ctrl_out=> Haspel_Li.st_ctrl.out);

		Haspel_Re.fb(
			t_wartezeit_bandende:= t#5s,
			b_bandende_Bandeinzug := ST_Bandwechsel_Kontroller.e_ls_bandende_re ,
			b_band_ok := gst_barcode_daten.b_band_rechts_ok AND gst_barcode_daten.b_band_ID_rechts_ok ,
			st_config:= Haspel_Re.fb.st_config,
			st_ctrl_in:= Haspel_Re.st_ctrl.in,
			st_visu := Haspel_Re.st_visu,
			st_zyl_heben:= zyl_haspel_re_heben,
			st_zyl_abspulen:= zyl_haspel_re_abspulen,
			st_zyl_sperren:= zyl_haspel_re_sperren,
			st_ctrl_out=> Haspel_Re.st_ctrl.out);

		IF gst_datensatz.st_md.b_auswahlSpruehoeler THEN
			ST_Menzel_Spruehoeler(
				st_config:= bandspruehoeler.st_config,
				st_ctrl_in:= bandspruehoeler.st_ctrl.in,
				lr_achse_position:= bestueckachse.NcToPlc.ModuloActPos,
				e_steuerung_ein:= ST_Safetyprogramm.se_steuerung_ein,
				e_druckwaechter:= ST_Betriebsfreigaben.e_druckwaechter,
				st_ctrl_out =>bandspruehoeler.st_ctrl.out,
				b_oelmangel=> ST_LampeMaterialMangel.b_materialmangel[1]);
		ELSE
			ST_BandoelerZylinder(
					st_config:= bandspruehoeler.st_config,
					st_ctrl_in:= bandspruehoeler.st_ctrl.in,
					lr_achse_position:= bestueckachse.NcToPlc.ModuloActPos,
					e_steuerung_ein:= ST_Safetyprogramm.se_steuerung_ein,
					e_druckwaechter:= ST_Betriebsfreigaben.e_druckwaechter,
					st_ctrl_out =>bandspruehoeler.st_ctrl.out,
					b_oelmangel=> ST_LampeMaterialMangel.b_materialmangel[1]);
		END_IF

		ST_Lesen_Schreiben_Tag(
			st_config:= Lesen_Schreiben_Tag.st_config,
			st_ctrl_in:= Lesen_Schreiben_Tag.st_ctrl.in,
			st_ctrl_out=> Lesen_Schreiben_Tag.st_ctrl.out);

		ST_Anwahl_Bandeinzug();
		ST_Scope();

	BESTUECKZELLE_1720:
		ST_AutoCheckIn( i_IntervalDay:=7 );
		ST_SaveAndLoad();
		ST_Datainit_Stationen();
		ST_Datainit_Achsen();

		ST_EthercatDiag();

		(* Grundmaschine *)
		EtherCatDiag[1]( );
		EtherCatDiag[1].st_config.b_station_aktiv := TRUE;

		(* Hublift links *)
		EtherCatDiag[2]( );
		EtherCatDiag[2].st_config.b_station_aktiv := gst_datensatz.st_md.b_hublift_links_aktiv;

		(* Hublift rechts *)
		EtherCatDiag[3]( );
		EtherCatDiag[3].st_config.b_station_aktiv := gst_datensatz.st_md.b_hublift_rechts_aktiv;

		(* Bandeinzug *)
		EtherCatDiag[4]( );
		EtherCatDiag[4].st_config.b_station_aktiv := NOT gst_datensatz.st_md.b_wt_transport_simulation;

		ST_UPS(st_config:= UPS.st_config,
			st_ctrl_in:= UPS.st_ctrl.in,
			b_Ups := TRUE,
			st_ctrl_out=> UPS.st_ctrl.out);

		ST_RoutingBackpanel(
			st_config:= routing_backpanel.st_config,
			st_ctrl_in:= routing_backpanel.st_ctrl.in,
			st_ctrl_out=> routing_backpanel.st_ctrl.out);

		ST_MotionFunctionPoints(
			st_ctrl_in:= edit_mfps.st_ctrl.in,
			st_ctrl_out=> edit_mfps.st_ctrl.out);

		ST_Schreibe_Persistente_Daten(
			bExecute:= ,
			bQuit:= ,
			t_schreibintervall:= t#60s,
			b_steuerung_ein:= ST_Safetyprogramm.se_steuerung_ein,
			bBusy=> ,
			bError=> ,
			nErrId=> );

		ST_System_DateAndTime();

		betriebsstundenzaehler.fb(
			b_eingekuppelt:= (ST_Z_Achse.fb_state_entry.i16_step > BEREIT AND ST_Z_Achse.fb_state_entry.i16_step < HALT) AND (gi16_betriebsart = AUTO),
			b_reset:= ,
			i32_betriebssekundenzaehler_in:= gst_datensatz.st_md.i32_betriebssekundenzaehler,
			i32_betriebssekundenzaehler=> gst_datensatz.st_md.i32_betriebssekundenzaehler);

		ST_Tuerverriegelung(
			e_quittiertaste:= ST_Safetyprogramm.se_quittiertaste);

		ST_LampeMaterialMangel(b_materialmangel:=  );

		ST_Zylinder();

		ST_start_OSK(bExecute:= ST_Safetyprogramm.se_quittiertaste);

		ST_Euchner_Handbedienpult();

		ST_TippTasten(
			i16_akt_stufe:= ,
			b_initialisierungsphase:= ,
			b_einfaedeln_aktiv:= ,
			st_visu:= visu,
			st_visu_hinten:= visu_hinten);

		ST_Betriebsarten(st_config:= betriebsarten.st_config);

		(* Übernahme der Daten aus der Datenbank: Beladen und Abgabe greifen dann auf diese Konfiguration zu *)
		wt_transport_kontroller.st_config.b_station_aktiv := gst_datensatz.st_md.b_wt_transport_aktiv;
		wt_transport_kontroller.st_config.b_station_in_simulation := gst_datensatz.st_md.b_wt_transport_simulation;

		ST_WT_Transport_Kontroller(
			st_config:= wt_transport_kontroller.st_config,
			st_ctrl_in:= wt_transport_kontroller.st_ctrl.in,
			st_visu:= visu,
			st_ctrl_out=> wt_transport_kontroller.st_ctrl.out);

		(* Aktivierung durch den Kontroller *)
		wt_transport_abgabe.st_config.b_station_aktiv := gst_datensatz.st_md.b_wt_transport_aktiv;
		wt_transport_abgabe.st_config.b_station_in_simulation := gst_datensatz.st_md.b_wt_transport_simulation;

		ST_WT_Transport_Abgabe(
			st_config:= wt_transport_abgabe.st_config,
			st_ctrl_in:= wt_transport_abgabe.st_ctrl.in,
			e_station_nachher_in_erlaubnis:= ,
			e_station_nachher_in_angekommen:= ,
			st_visu:= wt_transport_abgabe.st_visu,
			st_ctrl_out=> wt_transport_abgabe.st_ctrl.out,
			a_station_nachher_out_anforderung=> a_smema_station_nachher_out_anforderung,
			a_station_nachher_out_abgegeben=> a_smema_station_nachher_out_abgegeben);

		hublift_rechts.st_config.b_station_aktiv := gst_datensatz.st_md.b_hublift_rechts_aktiv;
		hublift_rechts.st_config.b_station_in_simulation := gst_datensatz.st_md.b_hublift_rechts_simulation;

		ST_Hublift_rechts(
			st_config:= hublift_rechts.st_config,
			st_ctrl_in:= hublift_rechts.st_ctrl.in,
			e_station_vorher_in_anforderung	:= ,
			e_station_vorher_in_abgegeben:= ,
			st_visu:= hublift_rechts.st_visu,
			st_ctrl_out=> hublift_rechts.st_ctrl.out,
			a_station_vorher_out_erlaubnis=> ,
			a_station_vorher_out_angekommen=> );
		IF hublift_rechts.st_config.b_station_aktiv OR hublift_rechts.st_config.b_station_in_simulation THEN
			ST_Hublift_rechts.e_station_vorher_in_abgegeben := ST_WT_Transport_Abgabe.a_station_nachher_out_abgegeben;
			ST_Hublift_rechts.e_station_vorher_in_anforderung := ST_WT_Transport_Abgabe.a_station_nachher_out_anforderung;
			ST_WT_Transport_Abgabe.e_station_nachher_in_angekommen := ST_Hublift_rechts.a_station_vorher_out_angekommen;
			ST_WT_Transport_Abgabe.e_station_nachher_in_erlaubnis := ST_Hublift_rechts.a_station_vorher_out_erlaubnis;
		ELSE
			ST_WT_Transport_Abgabe.e_station_nachher_in_angekommen := e_smema_station_nachher_in_angekommen;
			ST_WT_Transport_Abgabe.e_station_nachher_in_erlaubnis := e_smema_station_nachher_in_erlaubnis;
		END_IF

		balluff_tag_reader.fb(
			st_config:= balluff_tag_reader.fb.st_config,
			i16_addresse:= ,
			i16_anzahl_byte:= ,
			s_schreib_daten:= ,
			st_ctrl_in:= balluff_tag_reader.st_ctrl.in,
			s_lese_daten=> ,
			st_ctrl_out=> balluff_tag_reader.st_ctrl.out);

		barcode.fb(
			st_config:= barcode.fb.st_config,
			st_barcode_daten := gst_barcode_daten,
			b_steuerung_ein := ST_Safetyprogramm.se_steuerung_ein,
			b_bandende_links := ST_Bandeinzug_Kontroller_1720.e_ls_bandende_li ,
			b_bandende_rechts := ST_Bandeinzug_Kontroller_1720.e_ls_bandende_re,
			b_bandende_1720 := ST_Bandeinzug_Kontroller_1720.e_ls_bandende_li OR ST_Bandeinzug_Kontroller_1720.e_ls_bandende_re,
			b_band_nicht_gescannt=> ST_LampeMaterialMangel.b_materialmangel[5]);

		visu_hinten.in.bandfreigabe[0] := gst_barcode_daten.b_band_rechts_ok;
		visu_hinten.in.bandfreigabe[1] := gst_barcode_daten.b_band_links_ok;
		visu_hinten.in.band_ID[0] := gst_barcode_daten.b_band_ID_rechts_ok;
		visu_hinten.in.band_ID[1] := gst_barcode_daten.b_band_ID_links_ok;

		ST_VisuRouter();

		ST_Message_Produktion();

		ST_Bestueckachse(
			st_config_achse:= axis_bestueckachse.st_config,
			st_ctrl_in:= axis_bestueckachse.st_ctrl.in,
			e_steuerung_ein:= ST_Safetyprogramm.se_steuerung_ein,
			e_ba_mit_bedingungen:= ST_Safetyprogramm.se_ba_mit_bedingungen,
			e_tuere_vorne_offen:= ST_Safetyprogramm.se_tuere_vorne_offen,
			e_tuere_hinten_offen:= ST_Safetyprogramm.se_tuere_hinten_offen,
			st_visu:= axis_bestueckachse.st_visu,
			st_ctrl_out=> axis_bestueckachse.st_ctrl.out);

		ST_Z_Achse(
			st_config_achse:= axis_z_achse.st_config,
			st_ctrl_in:= axis_z_achse.st_ctrl.in,
			e_steuerung_ein:= ST_Safetyprogramm.se_steuerung_ein,
			e_ba_mit_bedingungen:= ST_Safetyprogramm.se_ba_mit_bedingungen,
			e_tuere_vorne_offen:= ST_Safetyprogramm.se_tuere_vorne_offen,
			e_tuere_hinten_offen:= ST_Safetyprogramm.se_tuere_hinten_offen,
			st_visu:= axis_z_achse.st_visu,
			st_ctrl_out=> axis_z_achse.st_ctrl.out,
			t_Z_Achse_ausfahren=>visu.ST_Service.t_Z_Achse_ausfahren,
			t_Bestueckung=>visu.ST_Service.t_Bestueckung,
			t_Z_Achse_einfahren=>visu.ST_Service.t_Z_Achse_einfahren);

		ST_TouchProbe();

		ST_Gesamthubzaehler();

		(* Aktivierung durch den Kontroller *)
		wt_transport_warteposition_1720.st_config.b_station_aktiv := gst_datensatz.st_md.b_wt_transport_aktiv;
		wt_transport_warteposition_1720.st_config.b_station_in_simulation := gst_datensatz.st_md.b_wt_transport_simulation;

		ST_WT_Transport_Warteposition_1720(
			st_config:= wt_transport_warteposition_1720.st_config,
			st_ctrl_in:= wt_transport_warteposition_1720.st_ctrl.in,
			e_station_vorher_in_anforderung	:= ,
			e_station_vorher_in_abgegeben:= ,
			st_visu:= wt_transport_warteposition_1720.st_visu,
			st_ctrl_out=> wt_transport_warteposition_1720.st_ctrl.out,
			a_station_vorher_out_erlaubnis=> a_smema_station_vorher_out_erlaubnis,
			a_station_vorher_out_angekommen=> a_smema_station_vorher_out_angekommen);

		(* Aktivierung durch den Kontroller *)
		wt_transport_beladen_1720.st_config.b_station_aktiv := gst_datensatz.st_md.b_wt_transport_aktiv;
		wt_transport_beladen_1720.st_config.b_station_in_simulation := gst_datensatz.st_md.b_wt_transport_simulation;

		ST_WT_Transport_Beladen_1720(
			st_config:= wt_transport_beladen_1720.st_config,
			st_ctrl_in:= wt_transport_beladen_1720.st_ctrl.in,
			st_visu:= wt_transport_beladen_1720.st_visu,
			st_ctrl_out=> wt_transport_beladen_1720.st_ctrl.out,
			t_WT_WechselZeit=>visu.ST_Service.t_WT_wechsel,
			t_traegerwechselzeit=>visu.ST_Service.t_traegerwechselzeit,
			t_Zentrierer_ausfahren=>visu.ST_Service.t_Zentrierer_ausfahren,
			t_Zentrierer_einfahren=>visu.ST_Service.t_Zentrierer_einfahren,
			t_komplett_zyklus=>visu.ST_Service.t_komplett_zyklus,);

		hublift_links.st_config.b_station_aktiv := gst_datensatz.st_md.b_hublift_links_aktiv;
		hublift_links.st_config.b_station_in_simulation := gst_datensatz.st_md.b_hublift_links_simulation;

		ST_Hublift_links(
			st_config:= hublift_links.st_config,
			st_ctrl_in:= hublift_links.st_ctrl.in,
			e_station_nachher_in_erlaubnis:= ,
			e_station_nachher_in_angekommen:= ,
			st_visu:= hublift_links.st_visu,
			st_ctrl_out=> hublift_links.st_ctrl.out,
			a_station_nachher_out_anforderung=> ,
			a_station_nachher_out_abgegeben=> );
		IF hublift_links.st_config.b_station_aktiv OR hublift_links.st_config.b_station_in_simulation THEN
			ST_Hublift_links.e_station_nachher_in_angekommen := ST_WT_Transport_Warteposition_1720.a_station_vorher_out_angekommen;
			ST_Hublift_links.e_station_nachher_in_erlaubnis := ST_WT_Transport_Warteposition_1720.a_station_vorher_out_erlaubnis;
			ST_WT_Transport_Warteposition_1720.e_station_vorher_in_abgegeben := ST_Hublift_links.a_station_nachher_out_abgegeben;
			ST_WT_Transport_Warteposition_1720.e_station_vorher_in_anforderung := ST_Hublift_links.a_station_nachher_out_anforderung;
		ELSE
			ST_WT_Transport_Warteposition_1720.e_station_vorher_in_abgegeben := e_smema_station_vorher_in_abgegeben;
			ST_WT_Transport_Warteposition_1720.e_station_vorher_in_anforderung := e_smema_station_vorher_in_anforderung;
		END_IF

		ST_Stoerungen_Quitt_1720(
			st_config:= stoerungen_quittieren.st_config,
			st_ctrl_in:= stoerungen_quittieren.st_ctrl.in,
			st_visu:= visu,
			st_visu_hinten:= visu_hinten,
			st_ctrl_out=> stoerungen_quittieren.st_ctrl.out,
			b_lampe_stoerung=> ST_Betriebsfreigaben.b_lampe_stoerung,
			b_lampe_produktion=> ST_Betriebsfreigaben.b_lampe_produktion);

		ST_Haspel_Kontroller_2H(
			t_abschaltzeit_motor:= haspel_kontroller.t_abschaltzeit_motor,
			b_drehrichtung_antrieb_links := gst_datensatz.st_wkz.b_laufrichtung_haspel_links,
			st_config:= haspel_kontroller.st_config,
			e_druckwaechter:= ST_Betriebsfreigaben.e_druckwaechter,
			e_steuerung_ein:= ST_Safetyprogramm.se_steuerung_ein,
			st_ctrl_in:= haspel_kontroller.st_ctrl.in,
			haspel1_ctrl_in:= haspel_li.st_ctrl.out,
			haspel2_ctrl_in:= haspel_re.st_ctrl.out,
			st_visu:= haspel_kontroller.st_visu,
			st_ctrl_out=> haspel_kontroller.st_ctrl.out,
			haspel1_ctrl_out=> haspel_li.st_ctrl.in,
			haspel2_ctrl_out=> haspel_re.st_ctrl.in,
			b_materialmangel_bandende=> ST_LampeMaterialMangel.b_materialmangel[0]);

		Haspel_Li.fb(
			t_wartezeit_bandende:= t#5s,
			b_bandende_Bandeinzug := ST_Bandwechsel_Kontroller.e_ls_bandende_li ,
			st_config:= Haspel_Li.fb.st_config,
			st_ctrl_in:= Haspel_Li.st_ctrl.in,
			st_visu := Haspel_Li.st_visu,
			st_zyl_heben:= zyl_haspel_li_heben,
			st_zyl_abspulen:= zyl_haspel_li_abspulen,
			st_zyl_sperren:= zyl_haspel_li_sperren,
			st_ctrl_out=> Haspel_Li.st_ctrl.out);

		Haspel_Re.fb(
			t_wartezeit_bandende:= t#5s,
			b_bandende_Bandeinzug := ST_Bandwechsel_Kontroller.e_ls_bandende_re ,
			st_config:= Haspel_Re.fb.st_config,
			st_ctrl_in:= Haspel_Re.st_ctrl.in,
			st_visu := Haspel_Re.st_visu,
			st_zyl_heben:= zyl_haspel_re_heben,
			st_zyl_abspulen:= zyl_haspel_re_abspulen,
			st_zyl_sperren:= zyl_haspel_re_sperren,
			st_ctrl_out=> Haspel_Re.st_ctrl.out);

		ST_Menzel_Spruehoeler(
			st_config:= bandspruehoeler.st_config,
			st_ctrl_in:= bandspruehoeler.st_ctrl.in,
			lr_achse_position:= bestueckachse.NcToPlc.ModuloActPos,
			e_steuerung_ein:= ST_Safetyprogramm.se_steuerung_ein,
			e_druckwaechter:= ST_Betriebsfreigaben.e_druckwaechter,
			st_ctrl_out =>bandspruehoeler.st_ctrl.out,
			b_oelmangel=> ST_LampeMaterialMangel.b_materialmangel[1]);

		ST_AbfallBlasluft(
			b_wkz_blasluft_aktiv:= gst_datensatz.st_wkz.b_wkz_blasluft_aktiv);

		ST_Lesen_Schreiben_Tag(
			st_config:= Lesen_Schreiben_Tag.st_config,
			st_ctrl_in:= Lesen_Schreiben_Tag.st_ctrl.in,
			st_ctrl_out=> Lesen_Schreiben_Tag.st_ctrl.out);

		ST_Anwahl_Bandeinzug();
		ST_Scope();

	RASTERFOLIE:
		ST_AutoCheckIn( i_IntervalDay:=7 );
		ST_SaveAndLoad();
		ST_Datainit_Stationen();
		ST_Datainit_Achsen();

		ST_EthercatDiag();

		(* Grundmaschine *)
		EtherCatDiag[1]( );
		EtherCatDiag[1].st_config.b_station_aktiv := TRUE;

		(* Hublift links *)
		EtherCatDiag[2]( );
		EtherCatDiag[2].st_config.b_station_aktiv := gst_datensatz.st_md.b_hublift_links_aktiv;

		(* Hublift rechts *)
		EtherCatDiag[3]( );
		EtherCatDiag[3].st_config.b_station_aktiv := gst_datensatz.st_md.b_hublift_rechts_aktiv;

		(* Bandeinzug *)
		EtherCatDiag[4]( );
		EtherCatDiag[4].st_config.b_station_aktiv := NOT gst_datensatz.st_md.b_wt_transport_simulation;

		ST_UPS(st_config:= UPS.st_config,
			st_ctrl_in:= UPS.st_ctrl.in,
			b_Ups := TRUE,
			st_ctrl_out=> UPS.st_ctrl.out);

		ST_RoutingBackpanel(
			st_config:= routing_backpanel.st_config,
			st_ctrl_in:= routing_backpanel.st_ctrl.in,
			st_ctrl_out=> routing_backpanel.st_ctrl.out);


		ST_MotionFunctionPoints(
			st_ctrl_in:= edit_mfps.st_ctrl.in,
			st_ctrl_out=> edit_mfps.st_ctrl.out);

		ST_Schreibe_Persistente_Daten(
			bExecute:= ,
			bQuit:= ,
			t_schreibintervall:= t#60s,
			b_steuerung_ein:= ST_Safetyprogramm.se_steuerung_ein,
			bBusy=> ,
			bError=> ,
			nErrId=> );

		ST_System_DateAndTime();

		betriebsstundenzaehler.fb(
			b_eingekuppelt:= (ST_Z_Achse.fb_state_entry.i16_step > BEREIT AND ST_Z_Achse.fb_state_entry.i16_step < HALT) AND (gi16_betriebsart = AUTO),
			b_reset:= ,
			i32_betriebssekundenzaehler_in:= gst_datensatz.st_md.i32_betriebssekundenzaehler,
			i32_betriebssekundenzaehler=> gst_datensatz.st_md.i32_betriebssekundenzaehler);

		ST_Tuerverriegelung(
			e_quittiertaste:= ST_Safetyprogramm.se_quittiertaste);

		ST_LampeMaterialMangel(b_materialmangel:=  );

		ST_Zylinder();

		ST_start_OSK(bExecute:= ST_Safetyprogramm.se_quittiertaste);

		ST_Euchner_Handbedienpult();

		ST_TippTasten(
			i16_akt_stufe:= ,
			b_initialisierungsphase:= ,
			b_einfaedeln_aktiv:= ,
			st_visu:= visu,
			st_visu_hinten:= visu_hinten);

		ST_Betriebsarten(st_config:= betriebsarten.st_config);

		(* Übernahme der Daten aus der Datenbank: Beladen und Abgabe greifen dann auf diese Konfiguration zu *)
		wt_transport_kontroller.st_config.b_station_aktiv := gst_datensatz.st_md.b_wt_transport_aktiv;
		wt_transport_kontroller.st_config.b_station_in_simulation := gst_datensatz.st_md.b_wt_transport_simulation;

		ST_WT_Transport_Kontroller(
			st_config:= wt_transport_kontroller.st_config,
			st_ctrl_in:= wt_transport_kontroller.st_ctrl.in,
			st_visu:= visu,
			st_ctrl_out=> wt_transport_kontroller.st_ctrl.out);

		(* Aktivierung durch den Kontroller *)
		wt_transport_abgabe.st_config.b_station_aktiv := gst_datensatz.st_md.b_wt_transport_aktiv;
		wt_transport_abgabe.st_config.b_station_in_simulation := gst_datensatz.st_md.b_wt_transport_simulation;

		ST_WT_Transport_Abgabe(
			st_config:= wt_transport_abgabe.st_config,
			st_ctrl_in:= wt_transport_abgabe.st_ctrl.in,
			e_station_nachher_in_erlaubnis:= ,
			e_station_nachher_in_angekommen:= ,
			st_visu:= wt_transport_abgabe.st_visu,
			st_ctrl_out=> wt_transport_abgabe.st_ctrl.out,
			a_station_nachher_out_anforderung=> a_smema_station_nachher_out_anforderung,
			a_station_nachher_out_abgegeben=> a_smema_station_nachher_out_abgegeben);

		hublift_rechts.st_config.b_station_aktiv := gst_datensatz.st_md.b_hublift_rechts_aktiv;
		hublift_rechts.st_config.b_station_in_simulation := gst_datensatz.st_md.b_hublift_rechts_simulation;

		ST_Hublift_rechts(
			st_config:= hublift_rechts.st_config,
			st_ctrl_in:= hublift_rechts.st_ctrl.in,
			e_station_vorher_in_anforderung	:= ,
			e_station_vorher_in_abgegeben:= ,
			st_visu:= hublift_rechts.st_visu,
			st_ctrl_out=> hublift_rechts.st_ctrl.out,
			a_station_vorher_out_erlaubnis=> ,
			a_station_vorher_out_angekommen=> );
		IF hublift_rechts.st_config.b_station_aktiv OR hublift_rechts.st_config.b_station_in_simulation THEN
			ST_Hublift_rechts.e_station_vorher_in_abgegeben := ST_WT_Transport_Abgabe.a_station_nachher_out_abgegeben;
			ST_Hublift_rechts.e_station_vorher_in_anforderung := ST_WT_Transport_Abgabe.a_station_nachher_out_anforderung;
			ST_WT_Transport_Abgabe.e_station_nachher_in_angekommen := ST_Hublift_rechts.a_station_vorher_out_angekommen;
			ST_WT_Transport_Abgabe.e_station_nachher_in_erlaubnis := ST_Hublift_rechts.a_station_vorher_out_erlaubnis;
		ELSE
			ST_WT_Transport_Abgabe.e_station_nachher_in_angekommen := e_smema_station_nachher_in_angekommen;
			ST_WT_Transport_Abgabe.e_station_nachher_in_erlaubnis := e_smema_station_nachher_in_erlaubnis;
		END_IF

		balluff_tag_reader.fb(
			st_config:= balluff_tag_reader.fb.st_config,
			i16_addresse:= ,
			i16_anzahl_byte:= ,
			s_schreib_daten:= ,
			st_ctrl_in:= balluff_tag_reader.st_ctrl.in,
			s_lese_daten=> ,
			st_ctrl_out=> balluff_tag_reader.st_ctrl.out);

		barcode.fb(
			st_config:= barcode.fb.st_config,
			st_barcode_daten := gst_barcode_daten,
			b_steuerung_ein := ST_Safetyprogramm.se_steuerung_ein,
			b_bandende_links := ST_Bandwechsel_Kontroller.e_ls_bandende_li ,
			b_bandende_rechts := ST_Bandwechsel_Kontroller.e_ls_bandende_re,
			b_bandende_1720 := ST_Bandeinzug_Kontroller_1720.e_ls_bandende_li,
			b_band_nicht_gescannt=> ST_LampeMaterialMangel.b_materialmangel[5]);

		visu_hinten.in.bandfreigabe[0] := gst_barcode_daten.b_band_rechts_ok;
		visu_hinten.in.bandfreigabe[1] := gst_barcode_daten.b_band_links_ok;
		visu_hinten.in.band_ID[0] := gst_barcode_daten.b_band_ID_rechts_ok;
		visu_hinten.in.band_ID[1] := gst_barcode_daten.b_band_ID_links_ok;

		ST_VisuRouter();

		ST_Message_Produktion();

 		ST_Rafl_Stoerungen_Quitt(
			st_config:= stoerungen_quittieren.st_config,
			st_ctrl_in:= stoerungen_quittieren.st_ctrl.in,
			st_visu:= visu,
			st_visu_hinten:= visu_hinten,
			st_ctrl_out=> stoerungen_quittieren.st_ctrl.out,
			b_lampe_stoerung=> ST_Betriebsfreigaben.b_lampe_stoerung,
			b_lampe_produktion=> ST_Betriebsfreigaben.b_lampe_produktion);

		ST_Rasterfolienmontage(
			st_config:= rasterfolienmontage.st_config,
			st_ctrl_in:= rasterfolienmontage.st_ctrl.in,
			st_visu:= rasterfolienmontage.st_visu,
			st_ctrl_out=> rasterfolienmontage.st_ctrl.out);

		ST_Rasterfolieneinzug(
			st_config:= rasterfolieneinzug.st_config,
			st_ctrl_in:= rasterfolieneinzug.st_ctrl.in,
			st_visu:= rasterfolieneinzug.st_visu,
			st_ctrl_out=> rasterfolieneinzug.st_ctrl.out);

		ST_Bestueckachse(
			st_config_achse:= axis_bestueckachse.st_config,
			st_ctrl_in:= axis_bestueckachse.st_ctrl.in,
			e_steuerung_ein:= ST_Safetyprogramm.se_steuerung_ein,
			e_ba_mit_bedingungen:= ST_Safetyprogramm.se_ba_mit_bedingungen,
			e_tuere_vorne_offen:= ST_Safetyprogramm.se_tuere_vorne_offen,
			e_tuere_hinten_offen:= ST_Safetyprogramm.se_tuere_hinten_offen,
			st_visu:= axis_bestueckachse.st_visu,
			st_ctrl_out=> axis_bestueckachse.st_ctrl.out);

		ST_Z_Achse(
			st_config_achse:= axis_z_achse.st_config,
			st_ctrl_in:= axis_z_achse.st_ctrl.in,
			e_steuerung_ein:= ST_Safetyprogramm.se_steuerung_ein,
			e_ba_mit_bedingungen:= ST_Safetyprogramm.se_ba_mit_bedingungen,
			e_tuere_vorne_offen:= ST_Safetyprogramm.se_tuere_vorne_offen,
			e_tuere_hinten_offen:= ST_Safetyprogramm.se_tuere_hinten_offen,
			st_visu:= axis_z_achse.st_visu,
			st_ctrl_out=> axis_z_achse.st_ctrl.out,
			t_Z_Achse_ausfahren=>visu.ST_Service.t_Z_Achse_ausfahren,
			t_Bestueckung=>visu.ST_Service.t_Bestueckung,
			t_Z_Achse_einfahren=>visu.ST_Service.t_Z_Achse_einfahren);

		ST_Y_Achse(
			st_config_achse:= axis_y_achse.st_config,
			st_ctrl_in:= axis_y_achse.st_ctrl.in,
			e_steuerung_ein:= ST_Safetyprogramm.se_steuerung_ein,
			e_ba_mit_bedingungen:= ST_Safetyprogramm.se_ba_mit_bedingungen,
			e_tuere_vorne_offen:= ST_Safetyprogramm.se_tuere_vorne_offen,
			e_tuere_hinten_offen:= ST_Safetyprogramm.se_tuere_hinten_offen,
			e_not_steu_tuer_schutz_ok:= ,
			st_visu:= axis_y_achse.st_visu,
			st_ctrl_out=> axis_y_achse.st_ctrl.out);

		ST_Gesamthubzaehler();

		(* Aktivierung durch den Kontroller *)
		wt_transport_beladen.st_config.b_station_aktiv := gst_datensatz.st_md.b_wt_transport_aktiv;
		wt_transport_beladen.st_config.b_station_in_simulation := gst_datensatz.st_md.b_wt_transport_simulation;

		ST_WT_Transport_Beladen(
			st_config:= wt_transport_beladen.st_config,
			st_ctrl_in:= wt_transport_beladen.st_ctrl.in,
			e_station_vorher_in_anforderung	:= ,
			e_station_vorher_in_abgegeben:= ,
			st_visu:= wt_transport_beladen.st_visu,
			st_ctrl_out=> wt_transport_beladen.st_ctrl.out,
			a_station_vorher_out_erlaubnis=> a_smema_station_vorher_out_erlaubnis,
			a_station_vorher_out_angekommen=> a_smema_station_vorher_out_angekommen,
			t_WT_WechselZeit=>visu.ST_Service.t_WT_wechsel,
			t_traegerwechselzeit=>visu.ST_Service.t_traegerwechselzeit,
			t_Zentrierer_ausfahren=>visu.ST_Service.t_Zentrierer_ausfahren,
			t_Zentrierer_einfahren=>visu.ST_Service.t_Zentrierer_einfahren,
			t_komplett_zyklus=>visu.ST_Service.t_komplett_zyklus,);

		hublift_links.st_config.b_station_aktiv := gst_datensatz.st_md.b_hublift_links_aktiv;
		hublift_links.st_config.b_station_in_simulation := gst_datensatz.st_md.b_hublift_links_simulation;

		ST_Hublift_links(
			st_config:= hublift_links.st_config,
			st_ctrl_in:= hublift_links.st_ctrl.in,
			e_station_nachher_in_erlaubnis:= ,
			e_station_nachher_in_angekommen:= ,
			st_visu:= hublift_links.st_visu,
			st_ctrl_out=> hublift_links.st_ctrl.out,
			a_station_nachher_out_anforderung=> ,
			a_station_nachher_out_abgegeben=> );
		IF hublift_links.st_config.b_station_aktiv OR hublift_links.st_config.b_station_in_simulation THEN
			ST_Hublift_links.e_station_nachher_in_angekommen := ST_WT_Transport_Beladen.a_station_vorher_out_angekommen;
			ST_Hublift_links.e_station_nachher_in_erlaubnis := ST_WT_Transport_Beladen.a_station_vorher_out_erlaubnis;
			ST_WT_Transport_Beladen.e_station_vorher_in_abgegeben := ST_Hublift_links.a_station_nachher_out_abgegeben;
			ST_WT_Transport_Beladen.e_station_vorher_in_anforderung := ST_Hublift_links.a_station_nachher_out_anforderung;
		ELSE
			ST_WT_Transport_Beladen.e_station_vorher_in_abgegeben := e_smema_station_vorher_in_abgegeben;
			ST_WT_Transport_Beladen.e_station_vorher_in_anforderung := e_smema_station_vorher_in_anforderung;
		END_IF

		ST_Lesen_Schreiben_Tag(
			st_config:= Lesen_Schreiben_Tag.st_config,
			st_ctrl_in:= Lesen_Schreiben_Tag.st_ctrl.in,
			st_ctrl_out=> Lesen_Schreiben_Tag.st_ctrl.out);

		ST_Anwahl_Bandeinzug();
		ST_Scope();

		ST_TouchProbe();

		ST_Haspel_Kontroller_2H(
			t_abschaltzeit_motor:= haspel_kontroller.t_abschaltzeit_motor,
			b_drehrichtung_antrieb_links := gst_datensatz.st_wkz.b_laufrichtung_haspel_links,
			st_config:= haspel_kontroller.st_config,
			e_druckwaechter:= ST_Betriebsfreigaben.e_druckwaechter,
			e_steuerung_ein:= ST_Safetyprogramm.se_steuerung_ein,
			st_ctrl_in:= haspel_kontroller.st_ctrl.in,
			haspel1_ctrl_in:= haspel_li.st_ctrl.out,
			haspel2_ctrl_in:= haspel_re.st_ctrl.out,
			st_visu:= haspel_kontroller.st_visu,
			st_ctrl_out=> haspel_kontroller.st_ctrl.out,
			haspel1_ctrl_out=> haspel_li.st_ctrl.in,
			haspel2_ctrl_out=> haspel_re.st_ctrl.in,
			b_materialmangel_bandende=> ST_LampeMaterialMangel.b_materialmangel[0]);

		Haspel_Li.fb(
			t_wartezeit_bandende:= t#5s,
			b_bandende_Bandeinzug := ST_Bandwechsel_Kontroller.e_ls_bandende_li ,
			b_band_ok := gst_barcode_daten.b_band_links_ok AND gst_barcode_daten.b_band_ID_links_ok,
			st_config:= Haspel_Li.fb.st_config,
			st_ctrl_in:= Haspel_Li.st_ctrl.in,
			st_visu := Haspel_Li.st_visu,
			st_zyl_heben:= zyl_haspel_li_heben,
			st_zyl_abspulen:= zyl_haspel_li_abspulen,
			st_zyl_sperren:= zyl_haspel_li_sperren,
			st_ctrl_out=> Haspel_Li.st_ctrl.out);

		Haspel_Re.fb(
			t_wartezeit_bandende:= t#5s,
			b_bandende_Bandeinzug := ST_Bandwechsel_Kontroller.e_ls_bandende_re ,
			b_band_ok := gst_barcode_daten.b_band_rechts_ok AND gst_barcode_daten.b_band_ID_rechts_ok ,
			st_config:= Haspel_Re.fb.st_config,
			st_ctrl_in:= Haspel_Re.st_ctrl.in,
			st_visu := Haspel_Re.st_visu,
			st_zyl_heben:= zyl_haspel_re_heben,
			st_zyl_abspulen:= zyl_haspel_re_abspulen,
			st_zyl_sperren:= zyl_haspel_re_sperren,
			st_ctrl_out=> Haspel_Re.st_ctrl.out);

END_CASE
END_PROGRAM

(* POU Maschine1700/WT Transport/ST_WT_Transport_Beladen_Achse_1700, ST *)
PROGRAM ST_WT_Transport_Beladen_Achse_1700
VAR_INPUT
	st_config								: struct_config;
	st_ctrl_in								: struct_ctrl_in;
	e_wt_im_aktionsfeld					: BOOL;
END_VAR
VAR_IN_OUT
	st_visu								: struct_visu;
END_VAR
VAR_OUTPUT
	st_ctrl_out							: struct_ctrl_out;
	t_WT_WechselZeit					: TIME := t#0ms;
	t_traegerwechselzeit					: TIME := t#0ms;
	t_Zentrierer_ausfahren					: TIME := t#0ms;
	t_Zentrierer_einfahren					: TIME := t#0ms;
	t_komplett_zyklus						: TIME := t#0ms;
END_VAR
VAR
	fb_ton_uez							: TON;
	fb_ton_wz							: TON;
	fb_ton_quitt							: TON;
	fb_ton_wt_auf_beladepos				: TON;
	fb_tof_wt_auf_beladepos				: TOF;
	fb_r_trig_start							: R_TRIG;
	fb_r_trig_beladepos					: R_TRIG;
	fb_r_trig_beladepos_verlassen			: R_TRIG;
	fb_state_entry							: ST_StateEntry;
	fb_traegerwechselzeit					: ST_Taktzeit;
	fb_WT_WechselZeit					: ST_Taktzeit;
	fb_Zentrierer_ausfahren				: ST_Taktzeit;
	fb_Zentrierer_einfahren					: ST_Taktzeit;
	t_bestueckzeit						: TIME := t#0ms;
	sm_wt_hat_beladepos_nicht_verlassen	: BOOL := FALSE;
	sm_tagnummer_ungueltig				: BOOL := FALSE;
	sm_wt_hat_kein_tag					: BOOL := FALSE;
	sm_tagreader_nicht_fertig				: BOOL := FALSE;
	sm_keine_bandfreigabe				: BOOL := FALSE;
	sm_sensorfehler_beladepos			: BOOL := FALSE;
	bm_abfrage_wt_auf_beladepos			: BOOL := FALSE;
	bm_abfrage_wt_auf_wartepos			: BOOL := FALSE;
	bm_warte_auf_wt_an_stopper			: BOOL := FALSE;
	bMerkerSchrittketteKommtVonInit		: BOOL := FALSE;
	fb_ton_abfrage_wt_auf_beladepos		: TON;
	fb_ton_warte_auf_wt_an_stopper			: TON;
	i									: INT := 0;

	(* zum Testen der Achsen nach Tausch, Bestückbild "Becherspucken", WKZ ausgebaut, Vorschubkontrolle abeschaltet,
	Bit muss von Programmierer geforct werden, zum Beenden Schlüsselschalter auf HAND und Zelle neu starten *)
	b_Dauertest_Achsen					: BOOL := FALSE;

	e_wt_auf_beladepos					AT %I* : BOOL;
	e_wt_beladepos_verlassen				AT %I* : BOOL;
	e_wt_auf_pufferstrecke					AT %I* : BOOL;
END_VAR
(* Zeiten *)
fb_ton_uez(IN:= , PT:= , Q=>  , ET=> );
fb_ton_wz(IN:= , PT:= , Q=> , ET=> );
fb_ton_quitt(IN:= , PT:= t#100ms, Q=> , ET=> );

fb_ton_wt_auf_beladepos(IN:= e_wt_im_aktionsfeld, PT:= t#200ms, Q=> , ET=> );
fb_tof_wt_auf_beladepos(IN:= e_wt_im_aktionsfeld, PT:= t#200ms, Q=> , ET=> );

(* Flanken *)
fb_r_trig_beladepos(CLK:= e_wt_auf_beladepos, Q=> );
fb_r_trig_beladepos_verlassen(CLK:= e_wt_beladepos_verlassen, Q=> );
fb_r_trig_start(CLK:= st_ctrl_in.b_start, Q=> );

(*Trägerwechselzeiten*)
fb_WT_WechselZeit(b_start:= , t_zeit=> );
fb_Zentrierer_ausfahren(b_start:= , t_zeit=> );
fb_Zentrierer_einfahren(b_start:= , t_zeit=> );

(* ==================================Toplevel=================================== *)
IF fb_state_entry.i16_next_step > INIT AND fb_state_entry.i16_next_step < FEHLER THEN
	(* Allgemeine Fehler *)
	IF st_ctrl_in.b_stop THEN
		fb_state_entry.i16_next_step := STOP;
	ELSIF zyl_wt_zentrierer_tisch.st_ctrl.out.b_fehler OR
		zyl_Indexier_Bestueckpos.st_ctrl.out.b_fehler THEN
		fb_state_entry.i16_next_step := FEHLER;
	(* Zylinder im Handbetrieb *)
	ELSIF gi16_betriebsart = HAND AND
		st_visu.st_zyl.i16_nr_zyl_im_handbetrieb = zyl_wt_zentrierer_tisch.fb.st_config.i16_identnummer OR
		st_visu.st_zyl.i16_nr_zyl_im_handbetrieb = zyl_Indexier_Bestueckpos.fb.st_config.i16_identnummer  THEN
		fb_state_entry.i16_next_step := FEHLER;
	END_IF
END_IF

(* ============================Haupt-Schrittkette================================ *)
fb_state_entry(
	i16_next_step:= ,
	i16_pos:= 1,
	s_debugtext:= ,
	E=> ,
	X=> ,
	i16_step=> ,
	i16_last_step=> );

CASE fb_state_entry.i16_step OF
(*=======================================================*)
	INIT_OBJ:
		IF st_config.b_config_fertig THEN
			fb_state_entry.i16_next_step := INIT;
		END_IF

